	//Условие перехода (20)→(21)
	//Последовательность "Переход К-М" завершена
	IF (K_M.finish) AND drm.timeout THEN
		drm.cmd := drm.error := 0; drm.timer_pt := cycle; drm.inc := FALSE; drm.step := 21;
		btn.K_M.cmd := FALSE; //Шаг проверки: Переход К-М // Кнопка "Переход К-М"
	END_IF;
21:	//Запись уставки таймера шага
	drm.step := 21;//Текущий шаг
	drm.timer_pt := cycle; //Таймер: один цикл вызова

	//Команды текущего шага
	(*1*) btn.NObs.cmd := drm.cmd.0 := drm.step_time <= cycle; //Шаг проверки: АОбс из Магистрали // Кнопка "НОбс"

	//Условие перехода (21)→(22)
	//Последовательность "НОбс" завершена
	IF (NObs.finish) AND drm.timeout THEN
		drm.cmd := drm.error := 0; drm.timer_pt := cycle; drm.inc := FALSE; drm.step := 22;
		btn.NObs.cmd := FALSE; //Шаг проверки: АОбс из Магистрали // Кнопка "НОбс"
	END_IF;
22:	//Запись уставки таймера шага
	drm.step := 22;//Текущий шаг
	drm.timer_pt := cycle; //Таймер: один цикл вызова

	//Команды текущего шага
	(*1*) btn.Bleeding.cmd := drm.cmd.0 := TRUE; //Шаг проверки: Стравливание из ГР под газом // Кнопка "Стравливание ЦБК"

	//Условие перехода (22)→(23)
	//Последовательность "Стравливание" завершена
	IF (Bleeding_full.finish) AND drm.timeout THEN
		drm.cmd := drm.error := 0; drm.timer_pt := cycle; drm.inc := FALSE; drm.step := 23;
		btn.Bleeding.cmd := FALSE; //Шаг проверки: Стравливание из ГР под газом // Кнопка "Стравливание ЦБК"
	END_IF;
23:	//Запись уставки таймера шага
	drm.step := 23;//Текущий шаг
	drm.timer_pt := 10; //Таймер: 10 секунд

	//Команды текущего шага
	(*1*) btn.Repair.cmd := drm.cmd.0 := drm.step_time <= cycle; //Шаг проверки: Переход в Ремонт // Кнопка "Ремонт"

	//Условие перехода (23)→(24)
	//Режим Ремонт
	IF (mde.Repair) AND drm.timeout THEN
		drm.cmd := drm.error := 0; drm.timer_pt := cycle; drm.inc := FALSE; drm.step := 24;
		btn.Repair.cmd := FALSE; //Шаг проверки: Переход в Ремонт // Кнопка "Ремонт"
	END_IF;
24:	//Запись уставки таймера шага
	drm.step := 24;//Текущий шаг
	drm.timer_pt := cycle; //Таймер: один цикл вызова

	//Команды текущего шага
	(*1*) finish := drm.cmd.0 := TRUE; //Завершение
	(*1*) drm.error.0 := NOT btn.test_off.out; //Нажмите кнопку "Комплексное тестирование отключить"

	//Условие перехода (24)→(0)
	//Кнопка "Комплексное тестирование отключить"
	IF (btn.test_off.out) AND drm.timeout THEN
		drm.cmd := drm.error := 0; drm.timer_pt := cycle; drm.inc := FALSE; drm.step := -1;
		finish := FALSE; //Завершение
	END_IF;
END_CASE

//Принудительный выход из последовательности
IF break THEN
	drm.step := -1; drm.cmd := drm.error := 0; drm.timer_pt := cycle; drm.inc := FALSE;
	init := FALSE; //Переинициализирование переменных
	btn.GR.cmd := FALSE; //Шаг проверки: ХП из ГР // Кнопка "ГР"
	btn.HP.cmd := FALSE; //Шаг проверки: ХП из ГР // Кнопка "ХП"
	btn.Start.cmd := FALSE; //Шаг проверки: ХП из ГР // Кнопка "Пуск"
	btn.KPK.cmd := FALSE; //Шаг проверки: КПК из ГР // Кнопка "КПК"
	btn.Start.cmd := FALSE; //Шаг проверки: КПК из ГР // Кнопка "Пуск"
	btn.APK.cmd := FALSE; //Шаг проверки: АПК из ГР под газом // Кнопка "АПК"
	btn.Start.cmd := FALSE; //Шаг проверки: АПК из ГР под газом // Кнопка "Пуск"
	btn.AOss.cmd := FALSE; //Шаг проверки: АОсс из Кольца // Кнопка "АОсс"
	btn.Unlock.cmd := FALSE; //Шаг проверки: АОсс из Кольца // Кнопка "Деблокировка"
	btn.GR.cmd := FALSE; //Шаг проверки: АПК из ГР без газа // Кнопка "ГР"
	btn.APK.cmd := FALSE; //Шаг проверки: АПК из ГР без газа // Кнопка "АПК"
	btn.Start.cmd := FALSE; //Шаг проверки: АПК из ГР без газа // Кнопка "Пуск"
	btn.NOss.cmd := FALSE; //Шаг проверки: НОсс из Кольца // Кнопка "НОсс"
	btn.GR.cmd := FALSE; //Шаг проверки: АПМ из ГР без газа // Кнопка "ГР"
	btn.AObs.cmd := FALSE; //Шаг проверки: АОбс из Магистрали // Кнопка "АОбс"
	btn.Unlock.cmd := FALSE; //Шаг проверки: АОбс из Магистрали // Кнопка "Деблокировка"
	btn.M_K.cmd := FALSE; //Шаг проверки: Переход М-К // Кнопка "Переход М-К"
	cmd_Nst_5000 := FALSE; //Шаг проверки: Повышение Nст до 5000 об/мин
	btn.K_M.cmd := FALSE; //Шаг проверки: Переход К-М // Кнопка "Переход К-М"
	btn.NObs.cmd := FALSE; //Шаг проверки: АОбс из Магистрали // Кнопка "НОбс"
	btn.Bleeding.cmd := FALSE; //Шаг проверки: Стравливание из ГР под газом // Кнопка "Стравливание ЦБК"
	btn.Repair.cmd := FALSE; //Шаг проверки: Переход в Ремонт // Кнопка "Ремонт"
	finish := FALSE; //Завершение
END_IF;

                  
END_FUNCTION_BLOCK

{region INFO}
(*
Назначение: Обновление настроек
Автор     : Дергаев
Дата      : 12.05.2025 16:11:36
Версия    : 00.01.00
*)
{endregion}
FUNCTION FuelRegTuns_update : BOOL
VAR_INPUT
END_VAR
VAR
END_VAR

                    FuelReg.limValUpNvd ();
FuelReg.limValUpNst ();
FuelReg.limValUpTst ();
FuelReg.limValUpTstStart();
FuelReg.limValUpPk ();
FuelReg.RegLimValUpNvd ();
FuelReg.RegLimValDnNvd ();
FuelReg.RegLimValUpNst ();
FuelReg.RegLimValUpTst ();
FuelReg.RegLimValUpTstStart();
FuelReg.RegLimValUpPk ();
FuelReg.ignitionStep ();
FuelReg.ignitionDelay ();
FuelReg.ignitionMaxTime ();
FuelReg.ignitionMaxVal ();
FuelReg.rateOnProg ();
FuelReg.stepOnProg ();
FuelReg.tau1vd ();
FuelReg.tau2vd ();
FuelReg.tau1st ();
FuelReg.tau2st();
FuelReg.tau1Tst ();
FuelReg.tau2Tst ();
FuelReg.tau1Pk ();
FuelReg.tau2Pk ();
FuelReg.dzVd ();
FuelReg.dzSt ();
FuelReg.dzTst ();
FuelReg.dzPk ();
FuelReg.kRVd ();
FuelReg.kLupVd ();
FuelReg.kLdnVd ();
FuelReg.kRst ();
FuelReg.kLupST ();
FuelReg.kLupTst ();
FuelReg.kLupPk ();
FuelReg. kCorrNvd();
FuelReg. kCorrNst();
FuelReg. kCorrTst();
FuelReg. kCorrPk ();
FuelReg.setNvdRegOn ();
FuelReg.setNvdStarterOff ();
FuelReg.setNvdHeat ();
FuelReg.setHeatTime ();
FuelReg.setNvdCool ();
FuelReg.setCoolTime ();
FuelReg.setDTign ();
FuelReg.dNvdUpLim();
FuelReg.dNvdDnLim();
FuelReg.dNstUpLim();
FuelReg.dTstUpLim();
FuelReg.dPkUpLim();
FuelReg.lowTonWork();
FuelReg.delayLowTonWork();
FuelReg.rateOnReg ();

                  
END_FUNCTION

// _^ - ^ _
// Автоматическая проверка защит
// Chekmarev

FUNCTION_BLOCK TAutoCheckShield
VAR_IN_OUT
	start	: BOOL;
END_VAR
VAR
	step	: INT := -1;
	// Проверяемые защиты ( FALSE - не проверена / не успех, TRUE - проверена )
	btn_AOss, 
	btn_AObs,
	AO_PRU,
	AO_BA,
	BEAO,
	SurgeD,
	Vs_D_Av,
	KPV2_wOpen,
	KPV4_wOpen,
	KPV15_wOpen,
	Nst_HH,
	Ntk_Av_HH,
	Nst_flt,
	Tg_inSt_HH,
	Fire_OD,
	Tg1_inSTdistort_HH,
	Tg_inSTflt,
	nIgnition,
	Fire_flt,
	Ntk_nBoost,
	DGdistort,
	Pa_out14_HH,
	BZA_ready_2,
	BZA_alr,
	Pm_TK_An,
	Pm_ST_An,
	Tm_outD_HH,
	Chip_outD,
	Ptg_inDG,
	Pm_Starter_Av,
	Pm_Starter_An,
	dP_F_Pv,
	Ptg_inTRK_LL,
	dPmg_LL,
	Pm_N_An,
	Zs_Nl,
	Kr6_OF_start,
	Causeless_KR1_OF,
	Causeless_KR2_OF,
	Causeless_KR6_OF,
	Causeless_KR10_11
			: BOOL;
			
	crsCurrent	: POINTER TO Tcrs;
	
	callCMD		: BOOL;
	timer		: TON; // Общий таймер
	wd			: TON; // злая собака
END_VAR

                    
IF start AND step = -1 THEN
	step := 5;
	start := FALSE;
	ELSE 
		start := FALSE;
END_IF

CASE step OF
	5:		// btn_AOss
		Reset();
		btn_AOss	:= FALSE;
		crsCurrent 	:= ADR ( crs.btn_AOss );
	6:
		APK_start( _time := T#15S, nextStep := step + 4, cmd := btn.AOss.cmd, checkCRS := btn_AOss );
		
	10:		// btn_AObs
		Reset();
		btn_AObs	:= FALSE;
		crsCurrent	:= ADR ( crs.btn_AObs );
	11:
		APK_start( _time := T#30S, nextStep := step + 4, cmd := btn.AObs.cmd, checkCRS := btn_AObs );
		
	15:		// AO_PRU
		Reset();
		AO_PRU		:= FALSE;
		crsCurrent	:= ADR ( crs.AO_PRU );
	16:
		APK_start( _time := T#29S, nextStep := step + 4, cmd := callCMD, checkCRS := AO_PRU );
		dipar.AO_PRU_1.sim_value := callCMD;
		dipar.AO_PRU_2.sim_value := callCMD;
		
	20:
		Reset();
		AO_BA		:= FALSE;
		crsCurrent	:= ADR ( crs.AO_BA );
	21:
		APK_start( _time := T#15S, nextStep := step + 4, cmd := dipar.AO_BA.sim_value, checkCRS := AO_BA );
		
	25:
		Reset();
		BEAO		:= FALSE;
		crsCurrent	:= ADR ( crs.BEAO );
	26:
		APK_start( _time := T#1S, nextStep := step + 4, cmd := dipar.BEAO.sim_value, checkCRS := BEAO );
		
	30:
		step := 31;
	31:
		step := step + 4;
		
	35:
		Reset();
		SurgeD		:= FALSE;
		crsCurrent	:= ADR ( crs.SurgeD );
	36:
		APK_start( _time := T#15S, nextStep := step + 4, cmd := dipar.SurgeD.sim_value, checkCRS := SurgeD );
		
	40:
		Reset();
		Vs_D_Av		:= FALSE;
		crsCurrent	:= ADR ( crs.Vs_D_Av );
	41:
		APK_start( _time := T#15S, nextStep := step + 4, cmd := dipar.Vs_D_Av.sim_value, checkCRS := Vs_D_Av );
		
	45:
		Reset();
		KPV2_wOpen:= FALSE;
		crsCurrent	:= ADR ( crs.KPV234_wOpen );
	46:
		APK_heat( _time := T#15S, nextStep := step + 4, cmd := callCMD, checkCRS := KPV2_wOpen );
		IF callCMD THEN
			dipar.KPV2_off.sim_value := FALSE;
		END_IF
		
	50: step := 51;		// KPV3
	51: step := 55;
	
	55: Reset();
		KPV4_wOpen	:= FALSE;
		crsCurrent	:= ADR ( crs.KPV234_wOpen );
	56: 
		APK_heat( _time := T#1M, nextStep := step + 4, cmd := callCMD, checkCRS := KPV4_wOpen );
		IF callCMD THEN
			dipar.KPV4_off.sim_value := FALSE;
		END_IF
		
	60:
		Reset();
		KPV15_wOpen	:= FALSE;
		crsCurrent	:= ADR ( crs.KPV15_wOpen );
	61:
		APK_work( _time := T#25S, nextStep := step + 4, cmd := callCMD, checkCRS := KPV15_wOpen );
		IF callCMD THEN
			dipar.KPV5_off.sim_value := FALSE;
		END_IF
		
	65:
		Reset();
		Nst_HH		:= FALSE;
		crsCurrent	:= ADR ( crs.Nst_HH );
	66:
		APK_start( _time := T#15S, nextStep := step + 4, cmd := callCMD, checkCRS := Nst_HH );
		acpar.Nst.sim_value := 9301 * TO_BYTE ( callCMD );
		acpar.Nst.sim_on	:= callCMD;
		
	70:
		Reset();
		Ntk_Av_HH	:= FALSE;
		crsCurrent	:= ADR ( crs.Ntk_Av_HH );
	71:
		APK_start( _time := T#15S, nextStep := step + 4, cmd := callCMD, checkCRS := Ntk_Av_HH );
		acpar.Ntk.sim_value := 8401 * TO_BYTE ( callCMD );	// aipar переписывается в ТР
		acpar.Ntk.sim_on	:= callCMD;		
		
	75:
		Reset();
		Nst_flt		:= FALSE;
		crsCurrent	:= ADR ( crs.Nst_flt );
	76:
		APK_start(_time := T#20S, nextStep := step + 4, cmd := callCMD, checkCRS := Nst_flt );
		aipar.Nst_1.flt_test	:= callCMD;
		aipar.Nst_2.flt_test	:= callCMD;
		
	80:
		Reset();
		Tg_inSt_HH	:= FALSE;
		crsCurrent	:= ADR ( crs.Tg_inST_HH );
	81:
		APK_start( _time := T#15S, nextStep := step + 4, cmd := callCMD, checkCRS := Tg_inSt_HH );
		acpar.Tg_inST.sim_value	:= 671 * TO_BYTE ( callCMD );
		acpar.Tg_inST.sim_on	:= callCMD;
		
	85:
		Reset();
		Fire_OD		:= FALSE;
		crsCurrent	:= ADR ( crs.Fire_OD );
	86:
		APK_start( _time := T#1S, nextStep := step + 4, cmd := dipar.Fire_OD.sim_value, checkCRS := Fire_OD );
		
	90:
		Reset();
		Tg1_inSTdistort_HH	:= FALSE;
		crsCurrent			:= ADR ( crs.Tg1_inSTdistort_HH );
	91:
		APK_heat(_time := T#30S, nextStep := step + 4, cmd := callCMD, checkCRS := Tg1_inSTdistort_HH );
		aipar.Tg_inST_1.sim_value := acpar.Tg_inST.value + 150 * TO_BYTE ( callCMD );
		
	95:
		Reset();
		Tg_inSTflt	:= FALSE;
		crsCurrent	:= ADR ( crs.Tg_inSTflt );
	96:
		APK_start( _time := T#10S, nextStep := step + 4, cmd := callCMD, checkCRS := Tg_inSTflt );
		aipar.Tg_inST_1.flt_test := callCMD;
		aipar.Tg_inST_3.flt_test := callCMD;
		aipar.Tg_inST_5.flt_test := callCMD;
		aipar.Tg_inST_6.flt_test := callCMD;
		
	100:
		Reset();
		nIgnition	:= FALSE;
		crsCurrent	:= ADR ( crs.nIgnition );		
	101:
		APK_start(_time := T#10S, nextStep := step + 4, cmd := callCMD, checkCRS := nIgnition );
		IF am.AZ.on AND callCMD THEN
			am.SK.on := FALSE;
		END_IF
	
	105:
		Reset();
		Fire_flt	:= FALSE;
		crsCurrent	:= ADR ( crs.Fire_flt );
	106:
		APK_work( _time := T#21S, nextStep := step + 4, cmd := callCMD, checkCRS := Fire_flt );
		crs.Tg1_inSTdistort_HH.alg_check := callCMD;
		crs.Tg2_inSTdistort_HH.alg_check := callCMD;
		crs.Tg3_inSTdistort_HH.alg_check := callCMD;
		crs.Tg4_inSTdistort_HH.alg_check := callCMD;
		crs.Tg5_inSTdistort_HH.alg_check := callCMD;
		crs.Tg6_inSTdistort_HH.alg_check := callCMD;
		acpar.Tg_inST.sim_on := callCMD;
		IF callCMD THEN
			acpar.Tg_inST.sim_value := acpar.Tg_inST.value - 10.0;
		END_IF
		
	110:
		Reset();
		Ntk_nBoost	:= FALSE;
		crsCurrent	:= ADR ( crs.Ntk_nBoost );
	111:
		APK_start( _time := T#30S, nextStep := step + 4, cmd := callCMD, checkCRS := Ntk_nBoost );
		acpar.Ntk.sim_on := callCMD AND aipar.Ntk_1.value > 5500;
		acpar.Nst.sim_on := callCMD AND aipar.Nst_1.value > 9100;
		acpar.Ntk.sim_value := 5500;
		acpar.Nst.sim_value := 9000;

	115:
		Reset();
		DGdistort	:= FALSE;
		crsCurrent	:= ADR ( crs.DGdistort );
	116:
		APK_heat( _time := T#10S, nextStep := step + 4, cmd := callCMD, checkCRS := DGdistort );
		aipar.DG_pos.sim_value := aopar.DG_set.value + 2 * TO_BYTE ( callCMD );
		
	120:
		Reset();
		Pa_out14_HH	:= FALSE;
		crsCurrent	:= ADR ( crs.Pa_out14_HH );
	121:
		APK_heat( _time := T#15S, nextStep := step + 4, cmd := callCMD, checkCRS := Pa_out14_HH );
		aipar.Pa_out14.sim_value := 2.1 * TO_BYTE ( callCMD );
		
	125:
		Reset();
		BZA_ready_2	:= FALSE;
		crsCurrent	:= ADR ( crs.BZA_ready_2 );
	126:
		APK_start( _time := T#1S, nextStep := step + 4, cmd := callCMD, checkCRS := BZA_ready_2 );
		IF callCMD THEN
			dipar.BZA_ready_2.sim_value := NOT callCMD;
		END_IF		
	
	130:
		Reset();
		BZA_alr		:= FALSE;
		crsCurrent	:= ADR ( crs.BZA_alr );
	131:
		APK_start( _time := T#45S, nextStep := step + 4, cmd := dipar.BZA_alr.sim_value, checkCRS := BZA_alr );
		
	135:
		Reset();
		Pm_TK_An	:= FALSE;
		crsCurrent	:= ADR ( crs.Pm_TK_An );
	136:
		APK_start( _time := T#1M, nextStep := step + 4, cmd := dipar.Pm_TK_An.sim_value, checkCRS := Pm_TK_An );
		
	140:
		Reset();
		Pm_ST_An	:= FALSE;
		crsCurrent	:= ADR ( crs.Pm_ST_An );
	141:
		APK_start( _time := T#70S, nextStep := step + 4, cmd := dipar.Pm_ST_An.sim_value, checkCRS := Pm_ST_An );
		
	145:
		Reset();
		Tm_outD_HH	:= FALSE;
		crsCurrent	:= ADR ( crs.Tm_outD_HH );
	146:
		APK_heat( _time := T#10S, nextStep := step + 4, cmd := callCMD, checkCRS := Tm_outD_HH );
		aipar.Tm_outD.sim_value	:= 86 * TO_BYTE ( callCMD );
		
	150:
		Reset();
		Chip_outD	:= FALSE;
		crsCurrent	:= ADR ( crs.Chip_outD );
	151:
		APK_start( _time := T#11S, nextStep := step + 4, cmd := dipar.Chip_outD.sim_value, checkCRS := Chip_outD );
		
	155:
		Reset();
		Ptg_inDG	:= FALSE;
		crsCurrent	:= ADR ( crs.Ptg_inDG_An );
	156:
		APK_start( _time := T#1M, nextStep := step + 4, cmd := dipar.Ptg_inDG_An.sim_value, checkCRS := Ptg_inDG );
		
	160:
		Reset();
		Pm_Starter_Av	:= FALSE;
		crsCurrent		:= ADR ( crs.Pm_Starter_Av );
	161:
		APK_start( _time := T#1M, nextStep := step + 4, cmd := callCMD, checkCRS := Pm_Starter_Av );
		dipar.Pm_Starter_Av.sim_value := callCMD;
	
	165:
		Reset();
		Pm_Starter_An	:= FALSE;
		crsCurrent		:= ADR ( crs.Pm_Starter_An );
	166:
		HP( _time := T#70S, nextStep := step + 4, cmd := callCMD, checkCRS := Pm_Starter_An );
		dipar.Pm_Starter_An.sim_value := callCMD;
		
	170:
		Reset();
		dP_F_Pv		:= FALSE;
		crsCurrent	:= ADR ( crs.dP_F_Pv );
	171:
		APK_start( _time := T#15S, nextStep := step + 4, cmd := dipar.dP_F_Pv.sim_value, checkCRS := dP_F_Pv );
	
	175:
		Reset();
		Ptg_inTRK_LL:= FALSE;
		crsCurrent	:= ADR ( crs.Ptg_inTRK_LL );
	176:
		APK_heat( _time := T#15S, nextStep := step + 4, cmd := callCMD, checkCRS := Ptg_inTRK_LL );
		IF callCMD THEN
			aipar.Ptg_inTRK.sim_value := 0.9;
		END_IF
		
	180:
		step := 181;
	181:
		step := step + 4;
		
	185:
		Reset();
		dPmg_LL		:= FALSE;
		crsCurrent	:= ADR ( crs.dPmg_LL );
	186:
		APK_start( _time := T#1M, nextStep := step + 4, cmd := callCMD, checkCRS := dPmg_LL );
		IF callCMD AND aipar.dPmg.value > 0.71 THEN
			aipar.dPmg.sim_value := 0.2;
		END_IF
		
	190:
		Reset();
		Pm_N_An		:= FALSE;
		crsCurrent	:= ADR ( crs.Pm_N_An );
	191:
		APK_start( _time := T#1M, nextStep := step + 4, cmd := dipar.Pm_N_An.sim_value, checkCRS := Pm_N_An );
	
	195:
		Reset();
		Zs_Nl		:= FALSE;
		crsCurrent	:= ADR ( crs.Zs_Nl );
	196:
		APK_start( _time := T#1M, nextStep := step + 4, cmd := dipar.Zs_Nl.sim_value, checkCRS := Zs_Nl );
		
	200:
		step := 201;
	201:
		step := step + 4;
	
	205:
		Reset();
		Kr6_OF_start	:= FALSE;
		crsCurrent		:= ADR ( crs.Kr6_off_start );
	206:
		APK_heat( _time := T#2M, nextStep := step + 4, cmd := callCMD, checkCRS := Kr6_OF_start );
		IF acpar.Nst.value > 300 THEN
			dipar.Kr6_off.sim_value := TRUE;
		END_IF
		
	210:
		Reset();
		Causeless_KR1_OF:= FALSE;
		crsCurrent		:= ADR ( crs.Causeless_KR1_off );
	211:
		APK_work( _time := T#1M, nextStep := step + 4, cmd := callCMD, checkCRS := Causeless_KR1_OF );
		IF callCMD THEN
			dipar.Kr1_ON.sim_value := NOT callCMD;
		END_IF
		
	215:
		Reset();
		Causeless_KR2_OF:= FALSE;
		crsCurrent		:= ADR ( crs.Causeless_KR2_off );
	216:
		APK_work( _time := T#1M, nextStep := step + 4, cmd := callCMD, checkCRS := Causeless_KR2_OF );
		IF callCMD THEN
			dipar.Kr2_ON.sim_value := NOT callCMD;
			dipar.Kr6_off.sim_value := callCMD;
		END_IF
		
	220:
		Reset();
		Causeless_KR6_OF := FALSE;
		crsCurrent		:= ADR ( crs.Causeless_KR6_off );
	221: 
		APK_work( _time := T#1M, nextStep := step + 4, cmd := callCMD, checkCRS := Causeless_KR6_OF );
		IF callCMD THEN
			dipar.Kr2_off.sim_value := callCMD;
			dipar.Kr6_ON.sim_value := NOT callCMD;
		END_IF
		
	225:
		Reset();
		Causeless_KR10_11:= FALSE;
		crsCurrent		:= ADR( crs.Causeless_KR10_11 );
	226:
		APK_start( _time := T#5M, nextStep := step + 4, cmd := callCMD, checkCRS := Causeless_KR10_11 );
		IF am.Kr15.on THEN
			dipar.Kr10_off.sim_value := FALSE;
		END_IF
		
	230:
		step := -1;
	
END_CASE

timer();
                  

ACTION Reset:
                        
timer ( IN := ( AOss.break XOR AOss.finish ) AND ( AObs.break XOR AObs.finish ) AND NOT timer.Q, PT := T#5S );
btn.Unlock.cmd 	:= timer.Q;
btn.GR.cmd		:= AOss.break AND aobs.break;
IF mde.GR THEN
	timer ( IN := FALSE );
	step := step + 1;
END_IF
wd ( IN := FALSE );
                      
END_ACTION

METHOD PRIVATE APK_start : BOOL
VAR_INPUT
	_time	: TIME;
	nextStep: INT;
END_VAR
VAR_IN_OUT
	cmd		: BOOL;
	checkCRS: BOOL;
END_VAR
                          IF mde.GR THEN
	timer (IN := TRUE, PT := T#5S);
	btn.APK.cmd := timer.Q;
END_IF
IF tch.ReadyAPK.value THEN
	timer ( IN := FALSE );
	btn.Unlock.cmd 	:= TRUE;
	btn.Start.cmd	:= TRUE;
END_IF
IF mde.APK THEN
	timer (IN := TRUE, PT := _time);
	cmd := timer.Q;
END_IF		
IF crsCurrent^.out THEN
	timer (IN 	:= FALSE);
	checkCRS 	:= TRUE;
	cmd			:= FALSE;
	step := nextStep;
	wd ( IN := FALSE );
END_IF

wd ( IN := TRUE, PT := T#5M + _time );
IF wd.Q THEN
	btn.AObs.cmd := TRUE;
	step 	:= nextStep;
	cmd		:= FALSE;
END_IF
                        
END_METHOD

METHOD PRIVATE APK_heat : BOOL
VAR_INPUT
	_time	: TIME;
	nextStep: INT;
END_VAR
VAR_IN_OUT
	cmd		: BOOL;
	checkCRS: BOOL;
END_VAR
                          IF mde.GR THEN
	timer (IN := TRUE, PT := T#5S);
	btn.APK.cmd := timer.Q;
END_IF
IF tch.ReadyAPK.value THEN
	timer (IN := FALSE);
	btn.Unlock.cmd 	:= TRUE;
	btn.Start.cmd	:= TRUE;
END_IF
IF tch.GTDHeat.value THEN
	timer (IN := TRUE, PT := _time);
	cmd := timer.Q;
END_IF		
IF crsCurrent^.out THEN
	timer (IN 	:= FALSE);
	checkCRS 	:= TRUE;
	cmd			:= FALSE;
	step := nextStep;
	wd ( IN := FALSE );
END_IF

wd ( IN := TRUE, PT := T#10M );
IF wd.Q THEN
	btn.AObs.cmd := TRUE;
	step 	:= nextStep;
	cmd		:= FALSE;
END_IF
                        
END_METHOD

METHOD PRIVATE APK_work : BOOL
VAR_INPUT
	_time	: TIME;
	nextStep: INT;
END_VAR
VAR_IN_OUT
	cmd		: BOOL;
	checkCRS: BOOL;
END_VAR
                          IF mde.GR THEN
	timer (IN := TRUE, PT := T#5S);
	btn.APK.cmd := timer.Q;
END_IF
IF tch.ReadyAPK.value THEN
	timer (IN := FALSE);
	btn.Unlock.cmd 	:= TRUE;
	btn.Start.cmd	:= TRUE;
END_IF
IF tch.GTDwork.value THEN
	timer (IN := TRUE, PT := _time);
	cmd := timer.Q;
END_IF		
IF crsCurrent^.out THEN
	timer (IN 	:= FALSE);
	checkCRS 	:= TRUE;
	cmd			:= FALSE;
	step := nextStep;
	wd ( IN := FALSE );
END_IF

wd ( IN := TRUE, PT := T#10M + _time );
IF wd.Q THEN
	btn.AObs.cmd := TRUE;
	step 	:= nextStep;
	cmd		:= FALSE;
END_IF
                        
END_METHOD

METHOD PRIVATE HP : BOOL
VAR_INPUT
	_time	: TIME;
	nextStep: INT;
END_VAR
VAR_IN_OUT
	cmd		: BOOL;
	checkCRS: BOOL;
END_VAR
                          IF mde.GR THEN
	timer (IN := TRUE, PT := T#5S);
	btn.HP.cmd := timer.Q;
END_IF
IF tch.ReadyHP.value THEN
	timer (IN := FALSE);
	btn.Unlock.cmd 	:= TRUE;
	btn.Start.cmd	:= TRUE;
END_IF
IF mde.HP THEN
	timer (IN := TRUE, PT := _time);
	cmd := timer.Q;
END_IF
IF crsCurrent^.out THEN
	timer (IN 	:= FALSE);
	checkCRS 	:= TRUE;
	cmd			:= FALSE;
	step := nextStep;
	wd ( IN := FALSE );
END_IF
wd ( IN := TRUE, PT := T#3M );
IF wd.Q THEN
	btn.AObs.cmd := TRUE;
	step 	:= nextStep;
	cmd		:= FALSE;
END_IF
                        
END_METHOD
END_FUNCTION_BLOCK

FUNCTION fun_ACS : BOOL
VAR_INPUT
END_VAR
VAR
END_VAR

                    ACS.ACS ( start := ACS.startACS );
                  
END_FUNCTION

{region INFO}
(*
 Назначение: Используется для присвоения переменным, предназначенным для передачи по МЭК-104 соответствующих значений
 Автор:      /Andrey/ 16.07.2025 17:15:07
*)
{endregion}
FUNCTION IEC104_update : BOOL
VAR_INPUT
END_VAR
VAR
END_VAR

                    //Режим/Тип:int4/Адрес:1
IEC104.GVL_mde_hmi_number.value := GVL.mde_hmi.number;
//Тест: пила, базовый цикл/Тип:REAL/Адрес:2
IEC104.test_Saw_Slow_value.value := test.Saw_Slow.value;
//Тест: пила, быстрый цикл/Тип:REAL/Адрес:3
IEC104.test_Saw_Fast_value.value := test.Saw_Fast.value;
//Тест: синус, базовый цикл/Тип:REAL/Адрес:4
IEC104.test_Sin_Slow_value.value := test.Sin_Slow.value;
//Частота вращения ротора ТК (1)/Тип:REAL/Адрес:5
IEC104.aipar_NTK_1_in_value.value := aipar.NTK_1.in_value;
//Частота вращения ротора ТК (2)/Тип:REAL/Адрес:6
IEC104.aipar_NTK_2_in_value.value := aipar.NTK_2.in_value;
//Частота вращения ротора СТ (1)/Тип:REAL/Адрес:7
IEC104.aipar_NST_1_in_value.value := aipar.NST_1.in_value;
//Частота вращения ротора СТ (2)/Тип:REAL/Адрес:8
IEC104.aipar_NST_2_in_value.value := aipar.NST_2.in_value;
//Положение дозирующей иглы ДУС/Тип:REAL/Адрес:9
IEC104.aipar_DG_Pos_in_value.value := aipar.DG_Pos.in_value;
//Давление воздуха за 14-й ступенью осевого компрессора/Тип:REAL/Адрес:10
IEC104.aipar_Pa_out14_in_value.value := aipar.Pa_out14.in_value;
//dP на конфузоре/Тип:REAL/Адрес:11
IEC104.aipar_dP_conf_in_value.value := aipar.dP_conf.in_value;
//Управление ТРК/Тип:REAL/Адрес:12
IEC104.aopar_DG_Set_value.value := aopar.DG_Set.value;
//СК закрыт/Тип:uint4/Адрес:13
IEC104.dipar_SK_off_status.value := dipar.SK_off.status;
//Открыть СК/Тип:uint4/Адрес:14
IEC104.dopar_SK_ON_status.value := dopar.SK_ON.status;
//диаг. (Сигнал управления положением дозатора газа)/Тип:REAL/Адрес:15
IEC104.aipar_DG_Pos_diag_in_value.value := aipar.DG_Pos_diag.in_value;
//Открыть КПВ1, 5/Тип:uint4/Адрес:16
IEC104.dopar_KPV15_ON_status.value := dopar.KPV15_ON.status;

                  
END_FUNCTION

{region INFO}
(*
 Назначение:   Ручной вызов обработчиков дискретных ИМов в base цикле
 Автор:        /chekmarev/ 17.04.2025
 Проект:       KA107
*)
{endregion}
FUNCTION am_update_base : BOOL
VAR
	KPV15du	: BOOL;
	KPV15on	: BOOL;
	KPV15off: BOOL;
	KPV23du	: BOOL;
	KPV23on	: BOOL;
	KPV23off: BOOL;
END_VAR

                    // ---------- блок самоподхвата ДУ у КПВ2 и КПВ3 по изменению одного из них с HMI
KPV23du	:= am.KPV2.cmd.0 OR am.KPV3.cmd.0;	// делаем так, чтобы не плодить глобальные переменные
KPV23on := am.KPV2.cmd.1 OR am.KPV3.cmd.1;
KPV23off := am.KPV2.cmd.2 OR am.KPV3.cmd.2;

engine.KPV2du( in	:= am.KPV2.cmd.0 );		// к этому моменту OPC сервер должен внести изменения в бит, если есть воздействие с HMI
engine.KPV2on( in	:= am.KPV2.cmd.1 );
engine.KPV2off( in	:= am.KPV2.cmd.2 );
engine.KPV3du( in	:= am.KPV3.cmd.0 );
engine.KPV3on( in	:= am.KPV3.cmd.1 );
engine.KPV3off( in	:= am.KPV3.cmd.2 );

IF engine.KPV2du.Qf OR engine.KPV3du.Qf THEN
	KPV23du := TRUE;
END_IF
IF engine.KPV2on.Qf OR engine.KPV3on.Qf THEN
	KPV23on := TRUE;
END_IF
IF engine.KPV2off.Qf OR engine.KPV3off.Qf THEN
	KPV23off := TRUE;
END_IF
IF engine.KPV2du.Qr OR engine.KPV3du.Qr THEN
	KPV23du	:= FALSE;
END_IF
IF engine.KPV2on.Qr OR engine.KPV3on.Qr THEN
	KPV23on := FALSE;
END_IF
IF engine.KPV2off.Qr OR engine.KPV3off.Qr THEN
	KPV23off := FALSE;
END_IF

// ---------- блок самоподхвата ДУ у КПВ1 и КПВ5 по изменению одного из них с HMI
KPV15du	:= am.KPV1.cmd.0 OR am.KPV5.cmd.0;
KPV15on	:= am.KPV1.cmd.1 OR am.KPV5.cmd.1;
KPV15off:= am.KPV1.cmd.2 OR am.KPV5.cmd.2;

engine.KPV1du( in	:= am.KPV1.cmd.0 );
engine.KPV1on( in	:= am.KPV1.cmd.1 );
engine.KPV1off( in	:= am.KPV1.cmd.2 );
engine.KPV5du( in	:= am.KPV5.cmd.0 );
engine.KPV5on( in	:= am.KPV5.cmd.1 );
engine.KPV5off( in	:= am.KPV5.cmd.2 );

IF engine.KPV1du.Qf OR engine.KPV5du.Qf THEN
	KPV15du := TRUE;
END_IF
IF engine.KPV1on.Qf OR engine.KPV5on.Qf THEN
	KPV15on := TRUE;
END_IF
IF engine.KPV1off.Qf OR engine.KPV5off.Qf THEN
	KPV15off := TRUE;
END_IF
IF engine.KPV1du.Qr OR engine.KPV5du.Qr THEN
	KPV15du	:= FALSE;
END_IF
IF engine.KPV1on.Qr OR engine.KPV5on.Qr THEN
	KPV15on := TRUE;
END_IF
IF engine.KPV1off.Qr OR engine.KPV5off.Qr THEN
	KPV15off := TRUE;
END_IF
// -----------------------------------

//КПВ 1
//Тип: 1x2
am.KPV1.cmd.0 	:= KPV15du;
am.KPV1.cmd.1 	:= KPV15on;
am.KPV1.cmd.2 	:= KPV15off;
am.KPV1(
	DU_prm := alg.V_000,
	onSigFlt := dipar.KPV1_ON.flt,
	onSig := dipar.KPV1_ON.value,
	onSig_sim_on := dipar.KPV1_ON.sim_on,
	onSig_sim_value := dipar.KPV1_ON.sim_value,
	offSigFlt := dipar.KPV1_off.flt,
	offSig := dipar.KPV1_off.value,
	offSig_sim_on := dipar.KPV1_off.sim_on,
	offSig_sim_value := dipar.KPV1_off.sim_value,
	onFlt := dopar.KPV15_ON.flt);
// dopar.KPV15_ON.value	-> Вызов в am_update_fast()	
//--------------------------------------------------------------------------

//КПВ 2
//Тип: 1x2
am.KPV2.cmd.0	:= KPV23du;
am.KPV2.cmd.1	:= KPV23on;
am.KPV2.cmd.2	:= KPV23off;
am.KPV2(
	DU_prm := alg.V_000,
	onSigFlt := dipar.KPV2_ON.flt,
	onSig := dipar.KPV2_ON.value,
	onSig_sim_on := dipar.KPV2_ON.sim_on,
	onSig_sim_value := dipar.KPV2_ON.sim_value,
	offSigFlt := dipar.KPV2_off.flt,
	offSig := dipar.KPV2_off.value,
	offSig_sim_on := dipar.KPV2_off.sim_on,
	offSig_sim_value := dipar.KPV2_off.sim_value,
	onFlt := dopar.KPV23_OFF.flt);
//--------------------------------------------------------------------------

//КПВ 3
//Тип: 1x2
am.KPV3.cmd.0	:= KPV23du;
am.KPV3.cmd.1	:= KPV23on;
am.KPV3.cmd.2	:= KPV23off;
am.KPV3(
	DU_prm := alg.V_000,
	onSigFlt := dipar.KPV3_ON.flt,
	onSig := dipar.KPV3_ON.value,
	onSig_sim_on := dipar.KPV3_ON.sim_on,
	onSig_sim_value := dipar.KPV3_ON.sim_value,
	offSigFlt := dipar.KPV3_off.flt,
	offSig := dipar.KPV3_off.value,
	offSig_sim_on := dipar.KPV3_off.sim_on,
	offSig_sim_value := dipar.KPV3_off.sim_value,
	onFlt := dopar.KPV23_OFF.flt);
dopar.KPV23_OFF.value := NOT am.KPV2.onOUT OR NOT am.KPV3.onOut;
//--------------------------------------------------------------------------

// КПВ4
// Штатный вызов (создан конфигуратором)

//КПВ 5
//Тип: 1x2
am.KPV5.cmd.0 := KPV15du;
am.KPV5.cmd.1 := KPV15on;
am.KPV5.cmd.2 := KPV15off;
am.KPV5(
	DU_prm := alg.V_000,
	onSigFlt := dipar.KPV5_ON.flt,
	onSig := dipar.KPV5_ON.value,
	onSig_sim_on := dipar.KPV5_ON.sim_on,
	onSig_sim_value := dipar.KPV5_ON.sim_value,
	offSigFlt := dipar.KPV5_off.flt,
	offSig := dipar.KPV5_off.value,
	offSig_sim_on := dipar.KPV5_off.sim_on,
	offSig_sim_value := dipar.KPV5_off.sim_value,
	onFlt := dopar.KPV15_ON.flt);
// dopar.KPV15_ON.value	-> Вызов в am_update_fast()
//--------------------------------------------------------------------------

//Кран 9
//Тип: 2x2
am.Kr9(
	DU_prm := FALSE,
	onSigFlt := dipar.Kr9_ON.flt,
	onSig := dipar.Kr9_ON.value,
	onSig_sim_on := dipar.Kr9_ON.sim_on,
	onSig_sim_value := dipar.Kr9_ON.sim_value,
	offSigFlt := dipar.Kr9_off.flt,
	offSig := dipar.Kr9_off.value,
	offSig_sim_on := dipar.Kr9_off.sim_on,
	offSig_sim_value := dipar.Kr9_off.sim_value,
	onFlt := dopar.Kr12_ON.flt,
	offFlt := dopar.KR12_OFF.flt);
	
//Кран 10
//Тип: 2x2
am.Kr10(
	DU_prm := FALSE,
	onSigFlt := dipar.Kr10_ON.flt,
	onSig := dipar.Kr10_ON.value,
	onSig_sim_on := dipar.Kr10_ON.sim_on,
	onSig_sim_value := dipar.Kr10_ON.sim_value,
	offSigFlt := dipar.Kr10_off.flt,
	offSig := dipar.Kr10_off.value,
	offSig_sim_on := dipar.Kr10_off.sim_on,
	offSig_sim_value := dipar.Kr10_off.sim_value,
	onFlt := dopar.Kr11_ON.flt,
	offFlt := dopar.Kr11_OFF.flt);
	
// ---------- блок самоподхвата ДУ у КПВ2 и КПВ3 по изменению одного из них с HMI
// выходы триггера сброшены, запоминаем текущее значение
engine.KPV2du( in	:= am.KPV2.cmd.0 );
engine.KPV2on( in	:= am.KPV2.cmd.1 );
engine.KPV2off( in	:= am.KPV2.cmd.2 );
engine.KPV3du( in	:= am.KPV3.cmd.0 );
engine.KPV3on( in	:= am.KPV3.cmd.1 );
engine.KPV3off( in	:= am.KPV3.cmd.2 );
// ------------------------------------
// ---------- блок самоподхвата ДУ у КПВ1 и КПВ5 по изменению одного из них с HMI
engine.KPV1du( in	:= am.KPV1.cmd.0 );
engine.KPV1on( in	:= am.KPV1.cmd.1 );
engine.KPV1off( in	:= am.KPV1.cmd.2 );
engine.KPV5du( in	:= am.KPV5.cmd.0 );
engine.KPV5on( in	:= am.KPV5.cmd.1 );
engine.KPV5off( in	:= am.KPV5.cmd.2 );
// -----------------------------------
                  
END_FUNCTION

FUNCTION AS_Link : BOOL
VAR_INPUT
END_VAR
VAR
END_VAR

                    s_tunpar.ASprot.Pin.value	:= aipar.Pg_inN.value; 
s_tunpar.ASprot.Pout.value	:= aipar.Pg_outN.value; 
s_tunpar.ASprot.Tin.value	:= aipar.Tg_inN.value;  
s_tunpar.ASprot.Tout.value	:= aipar.Tg_outN.value; 
s_tunpar.ASprot.dPconf.value:= aipar.dP_conf.value; 
s_tunpar.ASprot.Nst.value	:= acpar.Nst.value; 
s_tunpar.ASprot.Patm.value	:= 101.6; 

s_tunpar.ASprot.Pin.flt		:= aipar.Pg_inN.flt; 
s_tunpar.ASprot.Pout.flt	:= aipar.Pg_outN.flt; 
s_tunpar.ASprot.Tin.flt		:= aipar.Tg_inN.flt;  
s_tunpar.ASprot.Tout.flt	:= aipar.Tg_outN.flt; 
s_tunpar.ASprot.dPconf.flt	:= TRUE; //aipar.dP_conf.flt; 
s_tunpar.ASprot.Nst.flt		:= acpar.Nst.flt; 

s_tunpar_update();

s_tunpar.ASprot(
	cycle			:= cycle_time_fast, 
	D				:= 0.5917, // относительная плотность газа по воздуху - обычно выход блока расчета газовых констант, для упрощенного проекта задана постоянная
	mu				:= 17.091, // молярная масса газа, кг/кмоль - обычно выход блока расчета газовых констант, для упрощенного проекта задана постоянная
	sigDKS			:= FALSE, // при TRUE сигнал 
	sigPreSurgeOR	:= TRUE, // при TRUE сигнал предпомпажа (защиты) формируется при падении dPk ИЛИ росте Nst, при FALSE при падении dPk И росте Nst, проверить в работе
	protectOn		:= mde.M, // Взведение помпажной защиты. Магистраль? Переход К->М?
	sigCheck		:= mde.PZ, // Проверка защит 
	reset			:= btn.Unlock.out, // Деблокировка 
	calcSRon		:= TRUE,
	sigDKS 			:= TRUE,
	initSecResToMain := 3.0,
 	prod        => s_aspar.prod.value,  // объемная производительность, м3/с
 	prodCom     => s_aspar.prodCom.value, // коммерческая производительность, млн·нм3/сут
  	Qc          => s_aspar.Qc.value, // коммерческая производительность, нм3/ч
  	pressRatio  => s_aspar.pressRatio.value,
  	NstNorm     => s_aspar.NstNorm.value,
 // 	antisurgeBrk=> ,
 // 	mainContBrk => ,
 // 	res1ContBrk => ,
 // 	res2ContBrk => ,
  	surgeRes    => s_aspar.surgeRes.value,
  	ddPconf     => s_aspar.ddPconf.value, // производная перепада давления на конфузоре нагнетателя по времени
  	dNst        => s_aspar.dNst.value, // производная частоты вращения ротора нагнетателя по времени
  	preSurge    => tch.AS_preSurge.value, // сигнал "Предпомпажное состояние"
 	surge       => tch.AS_surge.value, // сигнал "Помпаж нагнетателя"
 // 	surgeAlertBrk=> , // сигнал "Отказ сигнализатора помпажа"
  	surgeSign_ddPconf=> tch.AS_surgeSign_ddPconf.value, // внутренний сигнал "Предпомпажное состояние" по падению dP на конфузоре //Dergaev 2024-11-02
  	surgeSign_dNst	=> tch.AS_surgeSign_dNst.value // внутренний сигнал "Предпомпажное состояние" по росту частоты вращения  //Dergaev 2024-11-02

//	emergOpenBypass=> Команда на 6 (вход в обработчик ИМ) - см. ALG_GO_AM
    
   );
   
 s_tunpar.ASprot.update();  
                  
END_FUNCTION

FUNCTION_BLOCK TASProtector
VAR_INPUT
// время цикла
  cycle : REAL;

// входные аналоговые параметры
  Pin    : Taspar; // P газа на входе ЦБК, МПа
  Pout   : Taspar; // P газа на выходе ЦБК, МПа
  Tin    : Taspar; // T газа на входе ЦБК, °С
  Tout   : Taspar; // T газа на выходе ЦБК, °С
  dPconf : Taspar; // перепад давления на конфузоре, кПа
  Nst    : Taspar; // Частота вращения СТ, об/мин
  Patm   : Taspar; // атмосферное давление, кПа
  
  D				: REAL; // относительная плотность газа по воздуху
  mu			: REAL; // молярная масса газа, кг/кмоль

  sigDKS        : BOOL; // работа на ДКС/линейной  КС
  sigPreSurgeOR : BOOL; // условие формировани¤ предпомпажного состо¤ни¤  
  protectOn 	: BOOL; // включить защиту
  sigCheck      : BOOL; // проверка защит
  reset			: BOOL; // сброс триггера открытия	
  check 		: BOOL; // проверка защит 
  calcSRon		: BOOL; // расчет помпажного запаса использовать
  initSecResToMain : REAL := 1.0; // начальное значение коэффициента пересчета второго контура в основной
END_VAR
VAR_OUTPUT
  prod        : REAL := 0.0 ; // объемная производительность, м3/с
  prodCom     : REAL := 0.0 ; // коммерческая производительность, млн·нм3/сут
  Qc          : REAL := 0.0 ; // коммерческая производительность, нм3/ч
  pressRatio  : REAL := 1.0 ;
  NstNorm     : REAL := 0.0 ;
  antisurgeBrk: BOOL := FALSE;
  mainContBrk : BOOL := false;
  res1ContBrk : BOOL := false;
  res2ContBrk : BOOL := false;
  surgeRes    : REAL := 100.0;
  ddPconf       : REAL; // производная перепада давления на конфузоре нагнетателя по времени
  dNst          : REAL; // производная частоты вращения ротора нагнетателя по времени
  preSurge      : BOOL; // сигнал "Предпомпажное состояние"
  surge         : BOOL; // сигнал "Помпаж нагнетателя"
  surgeAlertBrk : BOOL; // сигнал "Отказ сигнализатора помпажа"
  surgeSign_ddPconf : BOOL; // внутренний сигнал "Предпомпажное состояние" по падению dP на конфузоре //Dergaev 2024-11-02
  surgeSign_dNst	: BOOL; // внутренний сигнал "Предпомпажное состояние" по росту частоты вращения  //Dergaev 2024-11-02

  emergOpenBypass : BOOL; // команда экстренного открытия байпаса	
END_VAR
VAR
  resCalc      	: TSurgeResCalc; // блок расчета помпажного запаса
  surgeAlert   	: TSurgeAlert  ; // блок диагностики предпомпажного состояния
  init			: BOOL := TRUE; 	
END_VAR

                    
                  

METHOD update : BOOL
VAR_INPUT
END_VAR
                          // вычислить помпажный запас
resCalc(cycle  := cycle,
            Nst    := Nst.value,
            Pin    := Pin.value,
            Pout   := Pout.value,
            Tin    := Tin.value,
            dPconf := dPconf.value,
            Patm   := Patm.value,
            NstBrk    := Nst.flt,
            PinBrk    := Pin.flt,
            PoutBrk   := Pout.flt,
            dPconfBrk := dPconf.flt,
            c2Main := s_tunpar.c2Main.value,
            c1Main := s_tunpar.c1Main.value,
            c0Main := s_tunpar.c0Main.value,
            c21Res := s_tunpar.c2Res1.value,
            c11Res := s_tunpar.c1Res1.value,
            c01Res := s_tunpar.c0Res1.value,
            c22Res := s_tunpar.c2Res2.value,
            c12Res := s_tunpar.c1Res2.value,
            c02Res := s_tunpar.c0Res2.value,
            kConf  := s_tunpar.Kconf.value,
            nNorm  := s_tunpar.nNorm.value,
            D      := D,
            mu     := mu,
            check  := sigCheck,
			initSecResToMain := initSecResToMain,
			NstNorm=>NstNorm , 
			antisurgeBrk=>antisurgeBrk , 
			mainContBrk=>mainContBrk , 
			res1ContBrk=>res1ContBrk , 
			res2ContBrk=>res2ContBrk  );

IF protectOn THEN
	prod:=resCalc.prod; 
	prodCom:=resCalc.prodCom; 
	Qc:=resCalc.Qc; 
	pressRatio:=resCalc.pressRatio;
	surgeRes:=resCalc.surgeRes; 
ELSE
	prod:=0.0; 
	prodCom:=0.0; 
	Qc:=0.0; 
	pressRatio:=1.0; 			
	surgeRes:=100.0; 
END_IF;			
// обновить сигнализатор помпажа
surgeAlert( dPconf        := dPconf.value,
          	Nst           := Nst.value,
            dPconfBrk     := dPconf.flt,
          	NstBrk        := Nst.flt,
          	maxRateDPconf := s_tunpar.maxRateDPconf.value,
          	maxRateNst    := s_tunpar.maxRateNst.value,
          	SAoffDelay    := s_tunpar.SAoffDelay.value,
          	SAdelay       := s_tunpar.SAdelay.value,
          	blockDelay    := s_tunpar.blockDelay.value,
          	resetDelay    := s_tunpar.resetDelay.value,
          	cycle         := cycle,
          	permit        := protectOn,
          	alternate     := sigDKS,
          	preSurgeOR    := sigPreSurgeOR,
          	init          := init,
          	check         := sigCheck,
			ddPconf=>ddPconf , 
			dNst=>dNst , 
			preSurge=>preSurge , 
			surge=>surge , 
			surgeAlertBrk=>surgeAlertBrk , 
			surgeSign_ddPconf=>surgeSign_ddPconf , 
			surgeSign_dNst=>surgeSign_dNst );
			
IF init THEN init := FALSE; END_IF;			

// принудительное открытие байпаса
emergOpenBypass :=  protectOn AND NOT check AND ( surgeAlert.preSurge OR surgeAlert.surge OR calcSRon AND ( resCalc.surgeRes < s_tunpar.minSR.value ) OR emergOpenBypass ) AND NOT reset;
                        
END_METHOD
END_FUNCTION_BLOCK

{region INFO}
(*
Назначение: Числовые настройки
Автор     : Дергаев
Дата      : 20.03.2025 16:19:20
Версия    : 00.00.02
*)
{endregion}
FUNCTION s_tunpar_update : BOOL
VAR_INPUT
END_VAR
VAR
END_VAR

                    // код для функции обновления настроек
s_tunpar.c2Main(); // Коэфф. при 2-й степ. осн. системы координат
s_tunpar.c1Main(); // Коэфф. при 1-й степ. осн. системы координат
s_tunpar.c0Main(); // Коэфф. при 0-й степ. осн. системы координат
s_tunpar.c2Res1(); // Коэфф. при 2-й степ. 1-й рез. системы координат
s_tunpar.c1Res1(); // Коэфф. при 1-й степ. 1-й рез. системы координат
s_tunpar.c0Res1(); // Коэфф. при 0-й степ. 1-й рез. системы координат
s_tunpar.c2Res2(); // Коэфф. при 2-й степ. 2-й рез. системы координат
s_tunpar.c1Res2(); // Коэфф. при 1-й степ. 2-й рез. системы координат
s_tunpar.c0Res2(); // Коэфф. при 0-й степ. 2-й рез. системы координат
s_tunpar.minSR(); // Мин. помпажный запас
s_tunpar.maxPout (); // Макс. давление на выходе Н
s_tunpar.maxPR (); // Макс. степень сжатия
s_tunpar.Kconf(); // Коэффициент конфузора
s_tunpar.nNorm (); // Номинальная N СТ
s_tunpar.maxRateDPconf (); // Макс. ск. падения dP на конфузоре
s_tunpar.maxRateNst (); // Макс. ск. нарастания N СТ
s_tunpar.maxRateSR(); // Макс. ск. падения помпажного запаса
s_tunpar.maxRateSR_KM(); // Макс. ск. падения помпажного запаса К->М

                  
END_FUNCTION

FUNCTION handleMotoClock : BOOL

                    MotoClockGPA(
				start 	:= am.SK.on,
				stop	:= NOT am.SK.on,
				NO		:= alg.NO,
				AO		:= alg.AO,
				work	:= tch.GTDwork.value,
				reserve	:= alg.V_000,
				gaz		:= tch.Gas_N.value,
				
				countStart 	:= tunpar.countStart,
				countNO		:= tunpar.countNO,
				countAO		:= tunpar.countAO,
				generalOpTime	:= tunpar.generalOpTime,
				workOpTime		:= tunpar.workOpTime );
                  
END_FUNCTION

// Класс, обслуживающий наработку агрегата, а также подсчёт пуско-остановов
// Chekmarev
{attribute 'symbol' := 'none'}
FUNCTION_BLOCK TMotoClockHandler
VAR_INPUT
	start		: BOOL;		// сигнал пуска агрегата
	stop		: BOOL;		// сигнал останова двигателя
	NO			: BOOL;		// сигнал НО
	AO			: BOOL;		// сигнал АО
	work		: BOOL;		// агрегат в работе
	reserve		: BOOL;		// агрегат в резерве/ремонте
	gaz			: BOOL;		// газ в контуре
	path		: STRING := 'OpTime/engine/count.txt';	// путь до файла
END_VAR
VAR
	Qstart			: TEdgeDetect;
	Qno				: TEdgeDetect;
	Qao				: TEdgeDetect;
	
	// экземпляр ФБ для работы с файлом счётчиков пусков/остановов
	countFile	: FileManager;
	// ошибка работы с файлом
	err			: INT;
	init		: BOOL;
	// признак необходимости записи значений в файл
	xWrite		: BOOL;
	// признак пуска двигателя
	isStarted	: BOOL;
	// прежнее время
	oldTime		: UDINT;
	// временные переменные для хранения наработок
	generalOpTimeTemp,
	generalOpTimeOld,
	workOpTimeTemp,
	workOpTimeOld	: REAL;
END_VAR
VAR_IN_OUT
	// количество пусков
	countStart	: Ttunpar;
	// количество НО
	countNO		: Ttunpar;
	// количество АО
	countAO		: Ttunpar;

	// общая наработка в часах
	generalOpTime: Ttunpar;
	// наработка на режиме в часах
	workOpTime	: Ttunpar;
END_VAR
VAR CONSTANT
	rn	: STRING := '$R$N';
END_VAR

                    
Qstart( in := start );
Qno( in := NO );
Qao( in := AO );

IF Qstart.Qf THEN
	countStart.value := countStart.value + 1;
	xWrite := TRUE;
END_IF

IF Qno.Qr AND NOT AO THEN
	countNO.value	:= countNO.value + 1;
	xWrite := TRUE;
END_IF

IF Qao.Qf AND ( NOT reserve OR gaz ) THEN
	countAO.value	:= countAO.value + 1;
	xWrite := TRUE;
END_IF

IF NOT init THEN
	countFile.FileName := path;
	init := Read();
END_IF

IF xWrite THEN
	xWrite := NOT Write();
END_IF

countFile.Update();

isStarted := ( start OR isStarted ) AND NOT stop;
xWrite := OpTime();
                  

METHOD PRIVATE Write : BOOL
VAR
	temp	: STRING;
END_VAR
                          IF NOT countfile.xBusy THEN
	temp := CONCAT( TO_STRING( countStart.value ), rn );
	temp := CONCAT( temp, TO_STRING( countNO.value ));
	temp := CONCAT( temp, rn );
	temp := CONCAT( temp, TO_STRING( countAO.value ));
	temp := CONCAT( temp, rn );
	temp := CONCAT( temp, TO_STRING( generalOpTime.value ));
	temp := CONCAT( temp, rn );
	temp := CONCAT( temp, TO_STRING( workOpTime.value ));

	countFile.Record := temp;
END_IF

IF countFile.WDone THEN
	Write := TRUE;
END_IF

IF countFile.xError THEN
	err := countFile.eError;
	Write := TRUE;
END_IF
                        
END_METHOD

METHOD PRIVATE Read : BOOL
VAR
	temp	: STRING;
	sstart,
	sNO,
	sAO,
	sGeneral,
	sWork	: STRING;
	
	pos		: INT;
	l		: INT;
END_VAR
                          temp := countFile.Record;

IF countFile.RDone THEN
	pos		:= FIND( temp, rn ) - 1;
	sstart 	:= LEFT( temp, pos );
	pos 	:= pos + LEN( rn );
	temp	:= RIGHT( temp, LEN( temp ) - pos );
	pos 	:= FIND( temp , rn )- 1;
	sNO		:= LEFT( temp, pos );
	pos		:= pos + LEN( rn );
	temp	:= RIGHT( temp, LEN( temp ) - pos );
	pos		:= FIND( temp, rn ) - 1;
	sAO		:= LEFT( temp, pos );
	pos		:= pos + LEN( rn );
	temp	:= RIGHT( temp, LEN( temp ) - pos );
	pos		:= FIND( temp, rn ) - 1;
	sGeneral:= LEFT(temp, pos );
	pos		:= pos + LEN( rn );
	temp	:= RIGHT( temp, LEN( temp ) - pos );
	pos		:= FIND( temp, rn ) - 1;
	IF pos = -1 THEN
		pos := LEN( temp );
	END_IF
	sWork	:= LEFT(temp, pos );
	
	countStart.value	:= TO_REAL( sstart );
	countNO.value		:= TO_REAL( sNO );
	countAO.value		:= TO_REAL( sAO );
	
	generalOpTime.value	:= TO_REAL( sGeneral );
	workOpTime.value	:= TO_REAL( sWork );
	
	Read	:= TRUE;
END_IF

IF countFile.xError THEN
	err		:= countFile.eError;
	Read	:= TRUE;
END_IF
                        
END_METHOD

METHOD PRIVATE OpTime : BOOL
VAR
	cycle		: REAL;		// цикл вызова в часах
	currentTime	: UDINT;
END_VAR
VAR CONSTANT
	hour_ms	: REAL := 60_000.0 * 60.0;
END_VAR
                          currentTime	:= Util.SysTimeRtc.SysTimeGetMs();
cycle		:= TO_REAL( currentTime - oldTime ) / hour_ms;

generalOpTime.set_value	:= generalOpTime.value + cycle * TO_BYTE( isStarted );
workOpTime.set_value	:= workOpTime.value + cycle * TO_BYTE( work );

oldTime	:= Util.SysTimeRtc.SysTimeGetMs();
                        
END_METHOD
END_FUNCTION_BLOCK

// класс расчёта итоговой величина параметра по двум входным значениям
// Chekmarev 24.04.2025
//  0.0.01
// коэффициенты с 
FUNCTION_BLOCK TFreqRotorHandler
VAR_INPUT
	ch		: ARRAY[1..2] OF REAL; // измеряемые каналы
	minVal	: REAL	:= 100.0;
	maxVal	: REAL;
	flt_prm	: BOOL := TRUE;	// разрешение на расчёт неисправности
	disbal_Ch	: REAL := 100.0; // максимальный дисбаланс между каналами
	disbal_t: REAL	:= 0.16;// время расчёта дисбаланса, сек
	ucvV	: REAL	:= 500;	// максимальное изменение входной величины за цикл
	deblock	: BOOL;			// деблокировка
END_VAR
VAR_OUTPUT
	flt		: ARRAY[1..2] OF BOOL;	// отказ каналов по диапазону
	fltUcv	: ARRAY[1..2] OF BOOL;	// отказ каналов по скорости изменения
	disbal	: BOOL;
END_VAR
VAR_IN_OUT
	out		: Tacpar;
END_VAR
VAR
	oldVal	: ARRAY[1..2] OF REAL;
	disbalTmr	: TON;	// таймер дисбаланса
	ucvTmr		: ARRAY[1..2] OF TOF;	// таймеры удержки признака высокой скорости изменения
END_VAR
VAR CONSTANT
	ms_to_s	: UINT 	:= 1_000;
	PTucvTmr: TIME	:= T#30S;	// время удержания ПС по скорости изменения входного значения
END_VAR

                    flt_prm := flt_prm AND NOT deblock;

flt[1]	:= flt_prm AND ( ch[1] < minVal OR ch[1] > maxVal );
flt[2]	:= flt_prm AND ( ch[2] < minVal OR ch[2] > maxVal );

ucvTmr[1]( IN := flt_prm AND ABS( oldVal[1] - ch[1] ) > ucvV, PT := PTucvTmr );
ucvTmr[2]( IN := flt_prm AND ABS( oldVal[2] - ch[2] ) > ucvV, PT := PTucvTmr );

fltUcv[1] := ucvTmr[1].Q;
fltUcv[2] := ucvTmr[2].Q;

out.flt	:= ( flt[1] OR fltUcv[1] ) AND ( flt[2] OR fltUcv[2] );

IF ( ch[1] > ch[2] ) AND NOT ( flt[1] OR fltUcv[1] ) THEN
	out.in_value := ch[1];
	ELSIF NOT ( flt[2] OR fltUcv[2] ) THEN
	out.in_value := ch[2];
END_IF

disbalTmr (IN := flt_prm AND ( ABS( ch[1] - ch[2] ) > disbal_Ch ), PT := TO_TIME ( disbal_t * ms_to_s ));
disbal := disbalTmr.Q;

oldval[1] := ch[1];
oldVal[2] := ch[2];
                  
END_FUNCTION_BLOCK

// Контроль взвода защит на режимах
// Chekmarev
FUNCTION ShCntrl : BOOL
VAR
	shAlways	: BOOL;
	shInGas		: BOOL;
	shInWork	: BOOL;
	shOthers	: BOOL;
END_VAR

                    shAlways	:= 	crs.AO_BA.armed AND
				crs.AO_PRU.armed AND
				crs.AS_Av.armed AND
				crs.BEAO.armed AND
				crs.btn_AObs.armed AND
				crs.btn_AOss.armed AND
				crs.BZA_alr.armed AND
				crs.Chip_outD.armed AND
				crs.Fire_flt.armed AND
				crs.Fire_OD.armed AND
				crs.Nst_flt.armed AND
				crs.Nst_HH.armed AND
				crs.Ntk_Av_HH.armed AND
				crs.Ntk_flt.armed AND
				crs.Pa_out14_HH.armed  AND
				crs.SurgeD.armed AND
				crs.Tg_inST_HH.armed AND
				crs.Tg_inSTflt.armed AND
				crs.Tm_outD_HH.armed AND
				crs.Vs_D_Av.armed AND
				crs.Vsst_HH.armed AND
				crs.Vstk_HH.armed AND
				crs.Zs_Nl.armed ;
shInGas		:=	crs.dPmg_LL.armed AND tch.Gas_N.value OR NOT tch.Gas_N.value;
shInWork	:=( crs.Causeless_KR1_off.armed AND
				crs.Causeless_KR2_off.armed AND
				crs.Causeless_KR6_off.armed AND
				crs.KPV15_wOpen.armed AND 
				crs.Pm_ST_An.armed AND
				crs.Pm_TK_An.armed AND tch.GTDwork.value OR NOT tch.GTDwork.value ) AND
			  (	crs.Causeless_SK.armed AND
				crs.DGdistort.armed AND
				crs.KPV234_wOpen.armed AND
				crs.Pm_N_An.armed AND
				crs.Pm_SAR_An.armed AND
				crs.Ptg_inDG_An.armed AND
				crs.Ptg_inTRK_LL.armed AND
				crs.Tg1_inSTdistort_HH.armed AND
				crs.Tg2_inSTdistort_HH.armed AND
				crs.Tg3_inSTdistort_HH.armed AND
				crs.Tg4_inSTdistort_HH.armed AND
				crs.Tg5_inSTdistort_HH.armed AND
				crs.Tg6_inSTdistort_HH.armed AND ( tch.GTDHeat.value OR tch.GTDwork.value OR tch.GTDcool.value ) OR ( NOT tch.GTDHeat.value AND NOT tch.GTDwork.value AND NOT tch.GTDcool.value ));
shOthers	:=	crs.BZA_ready_2.armed AND
				crs.Causeless_KR10_11.armed AND
				crs.dP_F_Pv.armed AND
				crs.KPV15_nOpen.armed AND
				crs.Kr6_off_start.armed AND
				crs.nIgnition.armed AND	
				crs.Ntk_nBoost.armed AND
				crs.Pg_InKR13.armed AND
				crs.Pm_Starter_An.armed AND
				crs.Pm_Starter_Av.armed;

ShCntrl	:= shAlways AND shInGas AND shInWork;
                  
END_FUNCTION

PROGRAM PRG_IMIT
VAR
END_VAR

                    IF imitGPA.imit_on THEN
		GVL_IMIT.imitEngine(
		Tatm:= 15.0, 
		setDG1:= am.DG.set, 
		starter:= am.Kr11.isON AND am.Kr10.isOFF AND am.Kr13.on, 
		tuns:= ADR( GVL_IMIT.imitTuns ) 
		//posDG1=> , 
	);  
	
  	aipar.Ntk_1.sim_value := GVL_IMIT.imitEngine.Nvd;    
  	aipar.Ntk_2.sim_value := GVL_IMIT.imitEngine.Nvd;    
  	aipar.Nst_1.sim_value := GVL_IMIT.imitEngine.Nst;    
  	aipar.Nst_2.sim_value := GVL_IMIT.imitEngine.Nst;    
	aipar.Pa_out14.sim_value := GVL_IMIT.imitEngine.Pk;	
  	aipar.Tg_inST_1.sim_value := GVL_IMIT.imitEngine.Tst;  
  	aipar.Tg_inST_2.sim_value := GVL_IMIT.imitEngine.Tst;  
  	aipar.Tg_inST_3.sim_value := GVL_IMIT.imitEngine.Tst;  
  	aipar.Tg_inST_4.sim_value := GVL_IMIT.imitEngine.Tst;  
  	aipar.Tg_inST_5.sim_value := GVL_IMIT.imitEngine.Tst;  
  	aipar.Tg_inST_6.sim_value := GVL_IMIT.imitEngine.Tst;  
END_IF
                  
END_PROGRAM

PROGRAM HAND_DIAGN

                    UPD1_A1_1();
                  

ACTION UPD1_A1_1:
                        PsDiagn.PROXY_DI_16_012(MODULE := UPD1_A1_DI1, DATA := MODULE_UPD1_A1_DI1);
PsDiagn.PROXY_DI_16_012(MODULE := UPD1_A1_DI2, DATA := MODULE_UPD1_A1_DI2);
PsDiagn.PROXY_DI_16_012(MODULE := UPD1_A1_DI3, DATA := MODULE_UPD1_A1_DI3);
                      
END_ACTION
END_PROGRAM

{region INFO}
(*
 Назначение: Используется для сброса всех VAR_STAT сигнализаций
 Автор:  /Andrey/ 24.06.2025 16:50:31
 Версия: v00.00.22
 Проект: KA107__GPA2
*)
{endregion}
FUNCTION reset_alarm_var_stat : BOOL
VAR_INPUT
END_VAR

                    //Сбрасываем обобщенные сигнализации
//По типу и подсистемам в 0, потому что при сработке они выставляются в 1
crs.common.type_aggregated := crs.common.subsystem_aggregated := 0;
//По взводу защит все биты в 1, потому что при отсутствии взвода они сбрасываются в 0
crs.common.arm_aggregated := 16#FFFFFFFF;

//По типу биты 1-3 в 0 (для alr, lmt и trs, потому что при сработке они выставляются в 1), 4 и 5 в 1 (для ppu, потому что при сработке они сбрасываются в 0)
alr.common.type_aggregated := 2#110000;
//Для типов alr, lmt и trs по подсистемам все биты в 0, потому что при сработке они выставляются в 1
alr.common.subsystem_aggregated[1] := alr.common.subsystem_aggregated[2] := alr.common.subsystem_aggregated[3] := 0;
//Для ППУ по подсистемам все биты в 1, потому что при сработке они сбрасываются в 0
alr.common.subsystem_aggregated[4] := alr.common.subsystem_aggregated[5] := 16#FFFFFFFF;

                  
END_FUNCTION

{region INFO}
(*
 Назначение: Используется для сброса всех VAR_STAT входов/выходов
 Автор:  /Andrey/ 16.07.2025 17:15:05
 Версия: v00.00.01
 Проект: KA107
*)
{endregion}
FUNCTION reset_io_var_stat : BOOL
VAR_INPUT
END_VAR

                    //Сбрасываем для aipar
aipar.common.flt_aggregated := FALSE;
aipar.common.sim_aggregated := FALSE;
aipar.common.ucv_active := FALSE;

//Сбрасываем для aopar
aopar.common.flt_aggregated := FALSE;
aopar.common.sim_aggregated := FALSE;

//Сбрасываем для dipar
dipar.common.flt_aggregated := FALSE;
dipar.common.sim_aggregated := FALSE;

//Сбрасываем для dopar
dopar.common.flt_aggregated := FALSE;
dopar.common.sim_aggregated := FALSE;

                  
END_FUNCTION

{region INFO}
(*
 Назначение: Используется для сброса всех VAR_STAT ИМов
 Автор:  /Разработчик/ 08.08.2025 8:32:24
 Версия: v00.01.00
 Проект: KA107
*)
{endregion}
FUNCTION reset_am_var_stat : BOOL

                    am.common.flt_subsystem := 0;

                  
END_FUNCTION

// Используется для агрегации сигналов ИМов по подсистемам
FUNCTION aggregation_alarms : BOOL

                    
// crs
// Агрегация по типу
alg.AOss	:= crs.common.type_aggregated.1;
alg.AObs	:= crs.common.type_aggregated.2;


// ППУ
ppu.HR		:= ppu.common.type_aggregated.4;
ppu.GR		:= ppu.common.type_aggregated.5;

// Подсистемы
subsystem.EXT.aggregation_alarms( alr_common := alr.common, crs_common := crs.common );

subsystem.BD.aggregation_alarms( alr_common := alr.common, crs_common := crs.common );

subsystem.MSD.aggregation_alarms( alr_common := alr.common, crs_common := crs.common );

subsystem.VS.aggregation_alarms( alr_common := alr.common, crs_common := crs.common );

subsystem.AVOM.aggregation_alarms( alr_common := alr.common, crs_common := crs.common );

subsystem.BTG.aggregation_alarms( alr_common := alr.common, crs_common := crs.common );

subsystem.BPG.aggregation_alarms( alr_common := alr.common, crs_common := crs.common );

subsystem.POS.aggregation_alarms( alr_common := alr.common, crs_common := crs.common );

subsystem.BN.aggregation_alarms( alr_common := alr.common, crs_common := crs.common );

subsystem.BU.aggregation_alarms( alr_common := alr.common, crs_common := crs.common );

subsystem.GO.aggregation_alarms( alr_common := alr.common, crs_common := crs.common );
                  
END_FUNCTION

FUNCTION aggregation_am : BOOL

                    subsystem.EXT.AM_flt	:= am.common.flt_subsystem.1;

subsystem.BD.AM_flt		:= am.common.flt_subsystem.2;

subsystem.MSD.AM_flt	:= am.common.flt_subsystem.3;

subsystem.VS.AM_flt		:= am.common.flt_subsystem.4;

subsystem.AVOM.AM_flt	:= am.common.flt_subsystem.5;

subsystem.BTG.AM_flt	:= am.common.flt_subsystem.6;

subsystem.BPG.AM_flt	:= am.common.flt_subsystem.7;

subsystem.POS.AM_flt	:= am.common.flt_subsystem.8;

subsystem.BN.AM_flt		:= am.common.flt_subsystem.9;

subsystem.BU.AM_flt		:= am.common.flt_subsystem.10;

subsystem.GO.AM_flt		:= am.common.flt_subsystem.11;
                  
END_FUNCTION

FUNCTION ALG_BU_Link : BOOL

                    subsystem.BU();
                  
END_FUNCTION

FUNCTION ALG_VOU_Link : BOOL

                    subsystem.POS();
                  
END_FUNCTION

CONFIGURATION GPA2_SAU
  RESOURCE Application ON PLC
(* global variable list GVL_DIAGN *)
{attribute 'symbol' := 'readwrite'}
VAR_GLOBAL
	//Флаг активности ПЛК
	IS_ACTIVE: BOOL;
	//Активность ПЛК А
	IS_CPU_A: BOOL;
	//Активность ПЛК Б
	IS_CPU_B: BOOL;

	MODULE_UCP1_A1_ST1: PsDiagn.MODULE_ST_XX_X1X;
	MODULE_UCP1_A1_PP1: PsDiagn.MODULE_PP_00_XXX;
	MODULE_UCP1_A1_CU1: PsDiagn.MODULE_CU_XX_XXX;
	MODULE_UCP1_A1_FI1: PsDiagn.MODULE_DA_03_021_L_FRQ;
	MODULE_UCP1_A1_FI2: PsDiagn.MODULE_DA_03_021_L_FRQ;
	MODULE_UCP1_A1_AI1: PsDiagn.MODULE_AI_08_052;
	MODULE_UCP1_A1_AI2: PsDiagn.MODULE_AI_08_052;
	MODULE_UCP1_A1_AI3: PsDiagn.MODULE_AI_08_052;
	MODULE_UCP1_A1_AI4: PsDiagn.MODULE_AI_08_031;
	MODULE_UCP1_A1_AI5: PsDiagn.MODULE_AI_08_031;
	MODULE_UCP1_A1_AI6: PsDiagn.MODULE_AI_08_031;
	MODULE_UCP1_A1_AI7: PsDiagn.MODULE_AI_08_031;
	MODULE_UCP1_A1_ST2: PsDiagn.MODULE_ST_XX_X2X;
	MODULE_UCP1_A2_ST1: PsDiagn.MODULE_ST_XX_X1X;
	MODULE_UCP1_A2_PP1: PsDiagn.MODULE_PP_00_XXX;
	MODULE_UCP1_A2_AO1: PsDiagn.MODULE_AO_08_031;
	MODULE_UCP1_A2_DI1: PsDiagn.MODULE_AI_16_011;
	MODULE_UCP1_A2_DI2: PsDiagn.MODULE_AI_16_011;
	MODULE_UCP1_A2_DI3: PsDiagn.MODULE_DI_32_011;
	MODULE_UCP1_A2_DO1: PsDiagn.MODULE_DO_32_012;
	MODULE_UCP1_A2_DI4: PsDiagn.MODULE_DI_32_011;
	MODULE_UCP1_A2_ST2: PsDiagn.MODULE_ST_XX_X2X;
	MODULE_UE1_A1_ST1: PsDiagn.MODULE_ST_XX_X1X;
	MODULE_UE1_A1_PP1: PsDiagn.MODULE_PP_00_XXX;
	MODULE_UE1_A1_DI1: PsDiagn.MODULE_AI_16_011;
	MODULE_UE1_A1_DI2: PsDiagn.MODULE_AI_16_011;
	MODULE_UE1_A1_DI3: PsDiagn.MODULE_AI_16_011;
	MODULE_UE1_A1_DI4: PsDiagn.MODULE_DI_32_011;
	MODULE_UE1_A1_DI5: PsDiagn.MODULE_DI_32_011;
	MODULE_UE1_A1_DO1: PsDiagn.MODULE_DO_32_012;
	MODULE_UE1_A1_DI6: PsDiagn.MODULE_DI_32_011;
	MODULE_UE1_A1_DO2: PsDiagn.MODULE_DO_32_012;
	MODULE_UE1_A1_DI7: PsDiagn.MODULE_DI_32_011;
	MODULE_UE1_A1_ST2: PsDiagn.MODULE_ST_XX_X2X;
END_VAR
(* global variable list SETPOINTS_PERSISTENT_b9f40513_edea_4730_822c_5ab1a3caf7be *)
VAR_GLOBAL RETAIN PERSISTENT
	PERSISTENT_EXIST: BOOL;
END_VAR
(* global variable list alr *)
{region INFO}
(*
 Назначение: Признаки срабатывания предупредительных сигнализаций
 Автор:  /Andrey/ 24.06.2025 16:50:31
 Версия: v00.00.22
 Проект: KA107__GPA2
*)
{endregion}
{attribute 'qualified_only'}
{attribute 'symbol' := 'read'}
VAR_GLOBAL
	{attribute 'symbol' := 'none'}
	common : Talarm; //Общий сигнал для VAR_STAT

	{attribute 'export' := '("archive":"True","name":"Кнопка ЭАО на ПРУ нажата сигнал 1 (НР)","alarm":("type":"alr","action":"нет"),"condition":("set":"TRUE","reset":"FALSE","active":"dipar.EAO_PRU_1.value"))'}
	EAO_PRU_1 : Talarm:= (subsystem_num := 1, type_num := 1); //Кнопка ЭАО на ПРУ нажата сигнал 1 (НР)//DI/Внешние источники
	{attribute 'export' := '("archive":"True","name":"Кнопка ЭАО на ПРУ нажата сигнал 2 (НЗ)","alarm":("type":"alr","action":"нет"),"condition":("set":"TRUE","reset":"FALSE","active":"dipar.EAO_PRU_2.value"))'}
	EAO_PRU_2 : Talarm:= (subsystem_num := 1, type_num := 1); //Кнопка ЭАО на ПРУ нажата сигнал 2 (НЗ)//DI/Внешние источники
	{attribute 'export' := '("archive":"True","name":"Кнопка ЭАО на ПРУ нажата сигнал 3 (НЗ)","alarm":("type":"alr","action":"нет"),"condition":("set":"TRUE","reset":"FALSE","active":"dipar.EAO_PRU_3.value"))'}
	EAO_PRU_3 : Talarm:= (subsystem_num := 1, type_num := 1); //Кнопка ЭАО на ПРУ нажата сигнал 3 (НЗ)//DI/Внешние источники
	{attribute 'export' := '("archive":"True","name":"Нет связи с ПРУ","alarm":("type":"alr","action":"нет"),"condition":("set":"TRUE","reset":"FALSE","active":"NOT PRU.Link"))'}
	PRU_noLink : Talarm:= (subsystem_num := 1, type_num := 1, pt := t#1s0ms); //Нет связи с ПРУ//ALG/Внешние источники
	{attribute 'export' := '("archive":"True","name":"Загазованность контейнеров выше нормы","alarm":("type":"alr","action":"ХР"),"condition":("set":"TRUE","reset":"FALSE","active":"dipar.Zagaz_OD_Pv.value"))'}
	Zagaz_OD_Pv : Talarm:= (subsystem_num := 2, type_num := 1, pt := t#1s0ms); //Загазованность контейнеров выше нормы//DI/Блок двигателя
	{attribute 'export' := '("archive":"True","name":"Повышенная вибрация двигателя","alarm":("type":"alr","action":"нет"),"condition":("set":"TRUE","reset":"FALSE","active":"dipar.Vs_D_Pv.value"))'}
	Vs_D_Pv : Talarm:= (subsystem_num := 2, type_num := 1, pt := t#1s0ms); //Повышенная вибрация двигателя//DI/Блок двигателя
	{attribute 'export' := '("archive":"True","name":"Повыш. Вибрация ТК","alarm":("type":"alr","action":"нет"),"condition":("set":"TRUE","reset":"FALSE","active":"aipar.Vstk.setpoint.H"))'}
	Vstk_H : Talarm:= (subsystem_num := 2, type_num := 1, pt := t#1s0ms); //Повыш. Вибрация ТК//> 50/Блок двигателя
	{attribute 'export' := '("archive":"True","name":"Повыш. Вибрация СТ","alarm":("type":"alr","action":"нет"),"condition":("set":"TRUE","reset":"FALSE","active":"aipar.Vsst.setpoint.H"))'}
	Vsst_H : Talarm:= (subsystem_num := 2, type_num := 1, pt := t#1s0ms); //Повыш. Вибрация СТ//> 50/Блок двигателя
	{attribute 'export' := '("archive":"True","name":"Сигнализатор обледенения","alarm":("type":"alr","action":"ГР"),"condition":("set":"TRUE","reset":"FALSE","active":"dipar.Ace_alr.value"))'}
	Ace_alr : Talarm:= (subsystem_num := 2, type_num := 1, pt := t#1s0ms); //Сигнализатор обледенения//DI/Блок двигателя
	{attribute 'export' := '("archive":"True","name":"КПВ не открыты на пуске","alarm":("type":"alr","action":"нет"),"condition":("set":"acpar.Ntk.value > 2000 AND acpar.Ntk.value < 4500 AND alg.start","reset":"acpar.Ntk.value > 4500 OR alg.AO","active":"NOT ( dipar.KPV2_ON.value AND dipar.KPV3_ON.value AND dipar.KPV4_ON.value AND dipar.KPV1_ON.value AND dipar.KPV5_ON.value )"))'}
	KPV_nOpen : Talarm:= (subsystem_num := 2, type_num := 1, pt := t#1s0ms); //КПВ не открыты на пуске//DI/Блок двигателя
	{attribute 'export' := '("archive":"True","name":"КПВ234 не открыты","alarm":("type":"alr","action":"нет"),"condition":("set":"NOss.cmd_KPV234_On OR NObs.cmd_KPV234_On OR AOss.cmd_KPV234_On OR AObs.cmd_KPV234_On","reset":"acpar.Ntk.value < 2000","active":"NOT ( dipar.KPV2_ON.value AND dipar.KPV3_ON.value AND dipar.KPV4_ON.value )"))'}
	KPV234_nOpen : Talarm:= (subsystem_num := 2, type_num := 1, pt := t#1s0ms); //КПВ234 не открыты//ALG/Блок двигателя
	{attribute 'export' := '("archive":"True","name":"Повыш. Обороты СТ > 8500 об/мин","alarm":("type":"alr","action":"нет"),"condition":("set":"TRUE","reset":"FALSE","active":"acpar.Nst.setpoint.H"))'}
	Nst_H : Talarm:= (subsystem_num := 2, type_num := 1, pt := t#1s0ms); //Повыш. Обороты СТ > 8500 об/мин//> 8500 об/мин/Блок двигателя
	{attribute 'export' := '("archive":"True","name":"Высокая скорость изменения оборотов 1-ого канала ТК","alarm":("type":"alr","action":"нет"),"condition":("set":"TRUE","reset":"FALSE","active":"acpar_handler.handler.nTKcalc.fltUcv[1]"))'}
	Ntk_1_OV : Talarm:= (subsystem_num := 2, type_num := 1); //Высокая скорость изменения оборотов 1-ого канала ТК//ALG/Блок двигателя
	{attribute 'export' := '("archive":"True","name":"Высокая скорость изменения оборотов 2-ого канала ТК","alarm":("type":"alr","action":"нет"),"condition":("set":"TRUE","reset":"FALSE","active":"acpar_handler.handler.nTKcalc.fltUcv[2]"))'}
	Ntk_2_OV : Talarm:= (subsystem_num := 2, type_num := 1); //Высокая скорость изменения оборотов 2-ого канала ТК//ALG/Блок двигателя
	{attribute 'export' := '("archive":"True","name":"Значения оборотов 1-ого канала ТК не в диапазоне","alarm":("type":"alr","action":"нет"),"condition":("set":"TRUE","reset":"FALSE","active":"acpar_handler.handler.nTKcalc.flt[1]"))'}
	Ntk_1_UV : Talarm:= (subsystem_num := 2, type_num := 1); //Значения оборотов 1-ого канала ТК не в диапазоне//ALG/Блок двигателя
	{attribute 'export' := '("archive":"True","name":"Значения оборотов 2-ого канала ТК не в диапазоне","alarm":("type":"alr","action":"нет"),"condition":("set":"TRUE","reset":"FALSE","active":"acpar_handler.handler.nTKcalc.flt[2]"))'}
	Ntk_2_UV : Talarm:= (subsystem_num := 2, type_num := 1); //Значения оборотов 2-ого канала ТК не в диапазоне//ALG/Блок двигателя
	{attribute 'export' := '("archive":"True","name":"Значения оборотов 1-ого канала СТ не в диапазоне","alarm":("type":"alr","action":"нет"),"condition":("set":"TRUE","reset":"FALSE","active":"acpar_handler.handler.nSTcalc.flt[1]"))'}
	Nst_1_UV : Talarm:= (subsystem_num := 2, type_num := 1); //Значения оборотов 1-ого канала СТ не в диапазоне//ALG/Блок двигателя
	{attribute 'export' := '("archive":"True","name":"Значения оборотов 2-ого канала СТ не в диапазоне","alarm":("type":"alr","action":"нет"),"condition":("set":"TRUE","reset":"FALSE","active":"acpar_handler.handler.nSTcalc.flt[2]"))'}
	Nst_2_UV : Talarm:= (subsystem_num := 2, type_num := 1); //Значения оборотов 2-ого канала СТ не в диапазоне//ALG/Блок двигателя
	{attribute 'export' := '("archive":"True","name":"Высокая скорость изменения оборотов 1-ого канала СТ","alarm":("type":"alr","action":"нет"),"condition":("set":"TRUE","reset":"FALSE","active":"acpar_handler.handler.nSTcalc.fltUcv[1]"))'}
	Nst_1_OV : Talarm:= (subsystem_num := 2, type_num := 1); //Высокая скорость изменения оборотов 1-ого канала СТ//ALG/Блок двигателя
	{attribute 'export' := '("archive":"True","name":"Высокая скорость изменения оборотов 2-ого канала СТ","alarm":("type":"alr","action":"нет"),"condition":("set":"TRUE","reset":"FALSE","active":"acpar_handler.handler.nSTcalc.fltUcv[2]"))'}
	Nst_2_OV : Talarm:= (subsystem_num := 2, type_num := 1); //Высокая скорость изменения оборотов 2-ого канала СТ//ALG/Блок двигателя
	{attribute 'export' := '("archive":"True","name":"Повыш. Температура газа на входе СТ","alarm":("type":"alr","action":"нет"),"condition":("set":"TRUE","reset":"FALSE","active":"acpar.Tg_inST.setpoint.H"))'}
	Tg_inST_H : Talarm:= (subsystem_num := 2, type_num := 1); //Повыш. Температура газа на входе СТ//> 570 °С/Блок двигателя
	{attribute 'export' := '("archive":"True","name":"Нет сигнала: ТРК: готовность","alarm":("type":"alr","action":"ХР"),"condition":("set":"TRUE","reset":"FALSE","active":"NOT dipar.TRKready.value"))'}
	N_TRKready : Talarm:= (subsystem_num := 2, type_num := 1); //Нет сигнала: ТРК: готовность//Нет DI/Блок двигателя
	{attribute 'export' := '("archive":"True","name":"ТРК: авария","alarm":("type":"alr","action":"ХР"),"condition":("set":"TRUE","reset":"FALSE","active":"dipar.TRKalr.value"))'}
	TRKalr : Talarm:= (subsystem_num := 2, type_num := 1); //ТРК: авария//DI/Блок двигателя
	{attribute 'export' := '("archive":"True","name":"Контроль САУ не пройден","alarm":("type":"alr","action":"нет"),"condition":("set":"TRUE","reset":"FALSE","active":"check.tmrCancelPrm.Q"))'}
	nCheckSAU : Talarm:= (subsystem_num := 2, type_num := 1); //Контроль САУ не пройден//ALG/Блок двигателя
	{attribute 'export' := '("archive":"True","name":"Неисправность БЗА","alarm":("type":"alr","action":"нет"),"condition":("set":"tch.GTDWork.value","reset":"NOT tch.GTDWork.value","active":"NOT dipar.BZA_ready_1.value OR NOT dipar.BZA_ready_2.value"))'}
	BZA_flt : Talarm:= (subsystem_num := 2, type_num := 1); //Неисправность БЗА//ALG/Блок двигателя
	{attribute 'export' := '("archive":"True","name":"Пониж. Температура масла на входе двигателя","alarm":("type":"alr","action":"нет"),"condition":("set":"TRUE","reset":"FALSE","active":"aipar.Tm_inD.setpoint.L"))'}
	Tm_inD_L : Talarm:= (subsystem_num := 3, type_num := 1, pt := t#1s0ms); //Пониж. Температура масла на входе двигателя//< 40 °С/Маслосистема двигателя
	{attribute 'export' := '("archive":"True","name":"Уровень масла в МБД+Н минимальный","alarm":("type":"alr","action":"нет"),"condition":("set":"TRUE","reset":"FALSE","active":"dipar.Lm_MB_Pn.value"))'}
	Lm_MB_Pn : Talarm:= (subsystem_num := 3, type_num := 1, pt := t#1s0ms); //Уровень масла в МБД+Н минимальный//DI/Маслосистема двигателя
	{attribute 'export' := '("archive":"True","name":"Повыш. Температура масла на выходе АВОМД","alarm":("type":"alr","action":"нет"),"condition":("set":"TRUE","reset":"FALSE","active":"aipar.Tm_outAVOM.setpoint.H"))'}
	Tm_outAVOM_H : Talarm:= (subsystem_num := 5, type_num := 1, pt := t#1s0ms); //Повыш. Температура масла на выходе АВОМД//> 80 °С/Аппарат воздушного охлаждения масла двигателя
	{attribute 'export' := '("archive":"True","name":"Неисправность вентилятора 1 АВОМД","alarm":("type":"alr","action":"нет"),"condition":("set":"TRUE","reset":"FALSE","active":"am.Vn1_AVOM.flt"))'}
	Vn1_AVOM_flt : Talarm:= (subsystem_num := 5, type_num := 1, pt := t#1s0ms); //Неисправность вентилятора 1 АВОМД//DI/Аппарат воздушного охлаждения масла двигателя
	{attribute 'export' := '("archive":"True","name":"Неисправность вентилятора 2 АВОМД","alarm":("type":"alr","action":"нет"),"condition":("set":"TRUE","reset":"FALSE","active":"am.Vn2_AVOM.flt"))'}
	Vn2_AVOM_flt : Talarm:= (subsystem_num := 5, type_num := 1, pt := t#1s0ms); //Неисправность вентилятора 2 АВОМД//DI/Аппарат воздушного охлаждения масла двигателя
	{attribute 'export' := '("archive":"True","name":"Неисправность вентилятора 3 АВОМД","alarm":("type":"alr","action":"нет"),"condition":("set":"TRUE","reset":"FALSE","active":"am.Vn3_AVOM.flt"))'}
	Vn3_AVOM_flt : Talarm:= (subsystem_num := 5, type_num := 1, pt := t#1s0ms); //Неисправность вентилятора 3 АВОМД//DI/Аппарат воздушного охлаждения масла двигателя
	{attribute 'export' := '("archive":"True","name":"Неисправность вентилятора 4 АВОМД","alarm":("type":"alr","action":"нет"),"condition":("set":"TRUE","reset":"FALSE","active":"am.Vn4_AVOM.flt"))'}
	Vn4_AVOM_flt : Talarm:= (subsystem_num := 5, type_num := 1, pt := t#1s0ms); //Неисправность вентилятора 4 АВОМД//DI/Аппарат воздушного охлаждения масла двигателя
	{attribute 'export' := '("archive":"True","name":"Пониж. Давление топливного газа перед ТРК","alarm":("type":"alr","action":"нет"),"condition":("set":"alg.sh_TG","reset":"NOT alg.sh_TG","active":"aipar.Ptg_inTRK.setpoint.L"))'}
	Ptg_inTRK_L : Talarm:= (subsystem_num := 6, type_num := 1, pt := t#1s0ms); //Пониж. Давление топливного газа перед ТРК//< 20 кгс/см2/Блок топливного газа
	{attribute 'export' := '("archive":"True","name":"Повыш. Давление топливного газа перед ТРК","alarm":("type":"alr","action":"нет"),"condition":("set":"true","reset":"false","active":"aipar.Ptg_inTRK.setpoint.H"))'}
	Ptg_inTRK_H : Talarm:= (subsystem_num := 6, type_num := 1, pt := t#1s0ms); //Повыш. Давление топливного газа перед ТРК//> 27 кгс/см2/Блок топливного газа
	{attribute 'export' := '("archive":"True","name":"Давление газа перед дозатором газа Предупредительное","alarm":("type":"alr","action":"нет"),"condition":("set":"alg.sh_TG","reset":"NOT alg.sh_TG","active":"dipar.Ptg_inDG_Pn.value"))'}
	Ptg_inDG_Pn : Talarm:= (subsystem_num := 6, type_num := 1, pt := t#1s0ms); //Давление газа перед дозатором газа Предупредительное//DI/Блок топливного газа
	{attribute 'export' := '("archive":"True","name":"Перепад на сетке ВОУ","alarm":("type":"alr","action":"нет"),"condition":("set":"TRUE","reset":"FALSE","active":"dipar.Exh_VOU.value"))'}
	Exh_VOU : Talarm:= (subsystem_num := 8, type_num := 1, pt := t#1s0ms); //Перепад на сетке ВОУ//DI/Противообледенительная система и воздухоочистное устройство
	{attribute 'export' := '("archive":"True","name":"Опасность помпажа нагнетателя","alarm":("type":"alr","action":"нет"),"condition":("set":"TRUE","reset":"FALSE","active":"s_tunpar.ASprot.emergOpenBypass"))'}
	AS_Pv : Talarm:= (subsystem_num := 9, type_num := 1); //Опасность помпажа нагнетателя//ALG/Компрессорная установка/блок нагнетателя
	{attribute 'export' := '("archive":"True","name":"Пониж. Перепад давления “масло-газ”","alarm":("type":"alr","action":"нет"),"condition":("set":"alg.sh_dPmg","reset":"NOT alg.sh_dPmg","active":"aipar.dPmg.setpoint.L"))'}
	dPmg_L : Talarm:= (subsystem_num := 9, type_num := 1, pt := t#1s0ms); //Пониж. Перепад давления “масло-газ”//< 0.5 кгс/см2/Компрессорная установка/блок нагнетателя
	{attribute 'export' := '("archive":"True","name":"Уровень масла в МБУпл минимальный","alarm":("type":"alr","action":"нет"),"condition":("set":"TRUE","reset":"FALSE","active":"dipar.Lm_MBU_Pn.value"))'}
	Lm_MBU_Pn : Talarm:= (subsystem_num := 9, type_num := 1, pt := t#1s0ms); //Уровень масла в МБУпл минимальный//DI/Компрессорная установка/блок нагнетателя
	{attribute 'export' := '("archive":"True","name":"Повыш. Температура упорного подшипника Н","alarm":("type":"alr","action":"нет"),"condition":("set":"TRUE","reset":"FALSE","active":"aipar.Tup_N.setpoint.H"))'}
	Tup_N_H : Talarm:= (subsystem_num := 9, type_num := 1, pt := t#1s0ms); //Повыш. Температура упорного подшипника Н//> 80 °С/Компрессорная установка/блок нагнетателя
	{attribute 'export' := '("archive":"True","name":"Повыш. Температура опорного подшипника №1 Н","alarm":("type":"alr","action":"нет"),"condition":("set":"TRUE","reset":"FALSE","active":"aipar.Top_N_1.setpoint.H"))'}
	Top_N_1_H : Talarm:= (subsystem_num := 9, type_num := 1, pt := t#1s0ms); //Повыш. Температура опорного подшипника №1 Н//> 80 °С/Компрессорная установка/блок нагнетателя
	{attribute 'export' := '("archive":"True","name":"Повыш. Температура опорного подшипника №2 Н","alarm":("type":"alr","action":"нет"),"condition":("set":"TRUE","reset":"FALSE","active":"aipar.Top_N_2.setpoint.H"))'}
	Top_N_2_H : Talarm:= (subsystem_num := 9, type_num := 1, pt := t#1s0ms); //Повыш. Температура опорного подшипника №2 Н//> 80 °С/Компрессорная установка/блок нагнетателя
	{attribute 'export' := '("archive":"True","name":"Давление масла смазки Н предупредительная","alarm":("type":"alr","action":"нет"),"condition":("set":"NOT alg.V_000","reset":"alg.V_000","active":"dipar.Pm_N_Pn.value"))'}
	Pm_N_Pn : Talarm:= (subsystem_num := 9, type_num := 1, pt := t#1s0ms); //Давление масла смазки Н предупредительная//DI/Компрессорная установка/блок нагнетателя
	{attribute 'export' := '("archive":"True","name":"Нет сигнала: Предохранитель UCP1-XTFU1:1 питания модулей AO исправен","alarm":("type":"alr","action":"ХР"),"condition":("set":"TRUE","reset":"FALSE","active":"NOT dipar.Fuse_AO_UCP1.value"))'}
	N_Fuse_AO_UCP1 : Talarm:= (subsystem_num := 10, type_num := 1, pt := t#0s0ms); //Нет сигнала: Предохранитель UCP1-XTFU1:1 питания модулей AO исправен//Нет DI/Блок управления
	{attribute 'export' := '("archive":"True","name":"Нет сигнала: Предохранитель UCP1-XTFU1:2 питания модулей DO исправен","alarm":("type":"alr","action":"ХР"),"condition":("set":"TRUE","reset":"FALSE","active":"NOT dipar.Fuse_DO_UCP1.value"))'}
	N_Fuse_DO_UCP1 : Talarm:= (subsystem_num := 10, type_num := 1, pt := t#0s0ms); //Нет сигнала: Предохранитель UCP1-XTFU1:2 питания модулей DO исправен//Нет DI/Блок управления
	{attribute 'export' := '("archive":"True","name":"Нет сигнала: Предохранитель UCP1--XTFU6:1 питания датчиков температуры и влажности","alarm":("type":"alr","action":"ХР"),"condition":("set":"TRUE","reset":"FALSE","active":"NOT dipar.Fuse_Air_UCP1.value"))'}
	N_Fuse_Air_UCP1 : Talarm:= (subsystem_num := 10, type_num := 1, pt := t#0s0ms); //Нет сигнала: Предохранитель UCP1--XTFU6:1 питания датчиков температуры и влажности//Нет DI/Блок управления
	{attribute 'export' := '("archive":"True","name":"Нет сигнала: Предохранитель UE1-XTFU1:2 питания модулей DO исправен","alarm":("type":"alr","action":"ХР"),"condition":("set":"TRUE","reset":"FALSE","active":"NOT dipar.Fuse_DO_UE1.value"))'}
	N_Fuse_DO_UE1 : Talarm:= (subsystem_num := 10, type_num := 1, pt := t#0s0ms); //Нет сигнала: Предохранитель UE1-XTFU1:2 питания модулей DO исправен//Нет DI/Блок управления
	{attribute 'export' := '("archive":"True","name":"Перегрузка фильтра EV1 (Осн.)","alarm":("type":"alr","action":"ХР"),"condition":("set":"TRUE","reset":"FALSE","active":"dipar.EV1.value"))'}
	EV1 : Talarm:= (subsystem_num := 10, type_num := 1, pt := t#0s0ms); //Перегрузка фильтра EV1 (Осн.)//DI/Блок управления
	{attribute 'export' := '("archive":"True","name":"Перегрузка фильтра EV2 (Рез.)","alarm":("type":"alr","action":"ХР"),"condition":("set":"TRUE","reset":"FALSE","active":"dipar.EV2.value"))'}
	EV2 : Talarm:= (subsystem_num := 10, type_num := 1, pt := t#0s0ms); //Перегрузка фильтра EV2 (Рез.)//DI/Блок управления
	{attribute 'export' := '("archive":"True","name":"Нет сигнала: Контроль основного ввода питания (-KV1)","alarm":("type":"alr","action":"ХР"),"condition":("set":"TRUE","reset":"FALSE","active":"NOT dipar.U_main.value"))'}
	N_U_main : Talarm:= (subsystem_num := 10, type_num := 1, pt := t#0s0ms); //Нет сигнала: Контроль основного ввода питания (-KV1)//Нет DI/Блок управления
	{attribute 'export' := '("archive":"True","name":"Нет сигнала: Контроль резервного ввода питания (-KV2)","alarm":("type":"alr","action":"ХР"),"condition":("set":"TRUE","reset":"FALSE","active":"NOT dipar.U_res.value"))'}
	N_U_res : Talarm:= (subsystem_num := 10, type_num := 1, pt := t#0s0ms); //Нет сигнала: Контроль резервного ввода питания (-KV2)//Нет DI/Блок управления
	{attribute 'export' := '("archive":"True","name":"Контроль замыкания на землю питания PLC","alarm":("type":"alr","action":"нет"),"condition":("set":"TRUE","reset":"FALSE","active":"dipar.U_G_PLC.value"))'}
	U_G_PLC : Talarm:= (subsystem_num := 10, type_num := 1, pt := t#0s0ms); //Контроль замыкания на землю питания PLC//DI/Блок управления
	{attribute 'export' := '("archive":"True","name":"Контроль замыкания на землю питания AI","alarm":("type":"alr","action":"нет"),"condition":("set":"TRUE","reset":"FALSE","active":"dipar.U_G_AI.value"))'}
	U_G_AI : Talarm:= (subsystem_num := 10, type_num := 1, pt := t#0s0ms); //Контроль замыкания на землю питания AI//DI/Блок управления
	{attribute 'export' := '("archive":"True","name":"Контроль замыкания на землю питания DI","alarm":("type":"alr","action":"нет"),"condition":("set":"TRUE","reset":"FALSE","active":"dipar.U_G_DI.value"))'}
	U_G_DI : Talarm:= (subsystem_num := 10, type_num := 1, pt := t#0s0ms); //Контроль замыкания на землю питания DI//DI/Блок управления
	{attribute 'export' := '("archive":"True","name":"Контроль замыкания на землю питания БИЗ","alarm":("type":"alr","action":"нет"),"condition":("set":"TRUE","reset":"FALSE","active":"dipar.U_G_BIZ.value"))'}
	U_G_BIZ : Talarm:= (subsystem_num := 10, type_num := 1, pt := t#0s0ms); //Контроль замыкания на землю питания БИЗ//DI/Блок управления
	{attribute 'export' := '("archive":"True","name":"Нет сигнала: Контроль -AG1","alarm":("type":"alr","action":"ХР"),"condition":("set":"TRUE","reset":"FALSE","active":"NOT dipar.AG1.value"))'}
	N_AG1 : Talarm:= (subsystem_num := 10, type_num := 1, pt := t#0s0ms); //Нет сигнала: Контроль -AG1//Нет DI/Блок управления
	{attribute 'export' := '("archive":"True","name":"Нет сигнала: Контроль -AG2","alarm":("type":"alr","action":"ХР"),"condition":("set":"TRUE","reset":"FALSE","active":"NOT dipar.AG2.value"))'}
	N_AG2 : Talarm:= (subsystem_num := 10, type_num := 1, pt := t#0s0ms); //Нет сигнала: Контроль -AG2//Нет DI/Блок управления
	{attribute 'export' := '("archive":"True","name":"Нет сигнала: Контроль -AG3","alarm":("type":"alr","action":"ХР"),"condition":("set":"TRUE","reset":"FALSE","active":"NOT dipar.AG3.value"))'}
	N_AG3 : Talarm:= (subsystem_num := 10, type_num := 1, pt := t#0s0ms); //Нет сигнала: Контроль -AG3//Нет DI/Блок управления
	{attribute 'export' := '("archive":"True","name":"Нет сигнала: Контроль -AG4","alarm":("type":"alr","action":"ХР"),"condition":("set":"TRUE","reset":"FALSE","active":"NOT dipar.AG4.value"))'}
	N_AG4 : Talarm:= (subsystem_num := 10, type_num := 1, pt := t#0s0ms); //Нет сигнала: Контроль -AG4//Нет DI/Блок управления
	{attribute 'export' := '("archive":"True","name":"Нет сигнала: Контроль -AG9","alarm":("type":"alr","action":"ХР"),"condition":("set":"TRUE","reset":"FALSE","active":"NOT dipar.AG9.value"))'}
	N_AG9 : Talarm:= (subsystem_num := 10, type_num := 1, pt := t#0s0ms); //Нет сигнала: Контроль -AG9//Нет DI/Блок управления
	{attribute 'export' := '("archive":"True","name":"Нет сигнала: Контроль -AG10","alarm":("type":"alr","action":"ХР"),"condition":("set":"TRUE","reset":"FALSE","active":"NOT dipar.AG10.value"))'}
	N_AG10 : Talarm:= (subsystem_num := 10, type_num := 1, pt := t#0s0ms); //Нет сигнала: Контроль -AG10//Нет DI/Блок управления
	{attribute 'export' := '("archive":"True","name":"Нет сигнала: Контроль -AG15","alarm":("type":"alr","action":"ХР"),"condition":("set":"TRUE","reset":"FALSE","active":"NOT dipar.AG15.value"))'}
	N_AG15 : Talarm:= (subsystem_num := 10, type_num := 1, pt := t#0s0ms); //Нет сигнала: Контроль -AG15//Нет DI/Блок управления
	{attribute 'export' := '("archive":"True","name":"Нет сигнала: Контроль -AG16","alarm":("type":"alr","action":"ХР"),"condition":("set":"TRUE","reset":"FALSE","active":"NOT dipar.AG16.value"))'}
	N_AG16 : Talarm:= (subsystem_num := 10, type_num := 1, pt := t#0s0ms); //Нет сигнала: Контроль -AG16//Нет DI/Блок управления
	{attribute 'export' := '("archive":"True","name":"Нет сигнала: Контроль -AG5","alarm":("type":"alr","action":"ХР"),"condition":("set":"TRUE","reset":"FALSE","active":"NOT dipar.AG5.value"))'}
	N_AG5 : Talarm:= (subsystem_num := 10, type_num := 1, pt := t#0s0ms); //Нет сигнала: Контроль -AG5//Нет DI/Блок управления
	{attribute 'export' := '("archive":"True","name":"Нет сигнала: Контроль -AG6","alarm":("type":"alr","action":"ХР"),"condition":("set":"TRUE","reset":"FALSE","active":"NOT dipar.AG6.value"))'}
	N_AG6 : Talarm:= (subsystem_num := 10, type_num := 1, pt := t#0s0ms); //Нет сигнала: Контроль -AG6//Нет DI/Блок управления
	{attribute 'export' := '("archive":"True","name":"Нет сигнала: Контроль -AG8","alarm":("type":"alr","action":"ХР"),"condition":("set":"TRUE","reset":"FALSE","active":"NOT dipar.AG8.value"))'}
	N_AG8 : Talarm:= (subsystem_num := 10, type_num := 1, pt := t#0s0ms); //Нет сигнала: Контроль -AG8//Нет DI/Блок управления
	{attribute 'export' := '("archive":"True","name":"Нет сигнала: Контроль -AG17","alarm":("type":"alr","action":"ХР"),"condition":("set":"TRUE","reset":"FALSE","active":"NOT dipar.AG17.value"))'}
	N_AG17 : Talarm:= (subsystem_num := 10, type_num := 1, pt := t#0s0ms); //Нет сигнала: Контроль -AG17//Нет DI/Блок управления
	{attribute 'export' := '("archive":"True","name":"Нет сигнала: Контроль -AG18","alarm":("type":"alr","action":"ХР"),"condition":("set":"TRUE","reset":"FALSE","active":"NOT dipar.AG18.value"))'}
	N_AG18 : Talarm:= (subsystem_num := 10, type_num := 1, pt := t#0s0ms); //Нет сигнала: Контроль -AG18//Нет DI/Блок управления
	{attribute 'export' := '("archive":"True","name":"Нет сигнала: Контроль питания ПРУ","alarm":("type":"alr","action":"ХР"),"condition":("set":"TRUE","reset":"FALSE","active":"NOT dipar.U_PRU.value"))'}
	N_U_PRU : Talarm:= (subsystem_num := 10, type_num := 1, pt := t#0s0ms); //Нет сигнала: Контроль питания ПРУ//Нет DI/Блок управления
	{attribute 'export' := '("archive":"True","name":"Нет сигнала: Контроль питания ТРК осн.","alarm":("type":"alr","action":"ХР"),"condition":("set":"TRUE","reset":"FALSE","active":"NOT dipar.Utrk_main.value"))'}
	N_Utrk_main : Talarm:= (subsystem_num := 10, type_num := 1, pt := t#0s0ms); //Нет сигнала: Контроль питания ТРК осн.//Нет DI/Блок управления
	{attribute 'export' := '("archive":"True","name":"Контроль замыкания на землю питания ИМ","alarm":("type":"alr","action":"ХР"),"condition":("set":"TRUE","reset":"FALSE","active":"dipar.U_G_AM.value"))'}
	U_G_AM : Talarm:= (subsystem_num := 10, type_num := 1, pt := t#0s0ms); //Контроль замыкания на землю питания ИМ//DI/Блок управления
	{attribute 'export' := '("archive":"True","name":"Нет сигнала: Контроль питания AI","alarm":("type":"alr","action":"ХР"),"condition":("set":"TRUE","reset":"FALSE","active":"NOT dipar.U_AI.value"))'}
	N_U_AI : Talarm:= (subsystem_num := 10, type_num := 1, pt := t#0s0ms); //Нет сигнала: Контроль питания AI//Нет DI/Блок управления
	{attribute 'export' := '("archive":"True","name":"Нет сигнала: Контроль питания DI","alarm":("type":"alr","action":"ХР"),"condition":("set":"TRUE","reset":"FALSE","active":"NOT dipar.U_DI.value"))'}
	N_U_DI : Talarm:= (subsystem_num := 10, type_num := 1, pt := t#0s0ms); //Нет сигнала: Контроль питания DI//Нет DI/Блок управления
	{attribute 'export' := '("archive":"True","name":"Нет сигнала: Контроль питания БИЗ","alarm":("type":"alr","action":"ХР"),"condition":("set":"TRUE","reset":"FALSE","active":"NOT dipar.U_BIZ.value"))'}
	N_U_BIZ : Talarm:= (subsystem_num := 10, type_num := 1, pt := t#0s0ms); //Нет сигнала: Контроль питания БИЗ//Нет DI/Блок управления
	{attribute 'export' := '("archive":"True","name":"Нет сигнала: Контроль питания ИМ","alarm":("type":"alr","action":"ХР"),"condition":("set":"TRUE","reset":"FALSE","active":"NOT dipar.U_AM.value"))'}
	N_U_AM : Talarm:= (subsystem_num := 10, type_num := 1, pt := t#0s0ms); //Нет сигнала: Контроль питания ИМ//Нет DI/Блок управления
	{attribute 'export' := '("archive":"True","name":"Нет сигнала: Контроль питания аппаратуры вибрации, =24 В","alarm":("type":"alr","action":"ХР"),"condition":("set":"TRUE","reset":"FALSE","active":"NOT dipar.Uvs_24.value"))'}
	N_Uvs_24 : Talarm:= (subsystem_num := 10, type_num := 1, pt := t#0s0ms); //Нет сигнала: Контроль питания аппаратуры вибрации, =24 В//Нет DI/Блок управления
	{attribute 'export' := '("archive":"True","name":"Нет сигнала: Контроль питания дополнительного оборудования, =24В","alarm":("type":"alr","action":"ХР"),"condition":("set":"TRUE","reset":"FALSE","active":"NOT dipar.Uother_24.value"))'}
	N_Uother_24 : Talarm:= (subsystem_num := 10, type_num := 1, pt := t#0s0ms); //Нет сигнала: Контроль питания дополнительного оборудования, =24В//Нет DI/Блок управления
	{attribute 'export' := '("archive":"True","name":"Нет сигнала: Контроль питания ИМ2","alarm":("type":"alr","action":"ХР"),"condition":("set":"TRUE","reset":"FALSE","active":"NOT dipar.U_AM2.value"))'}
	N_U_AM2 : Talarm:= (subsystem_num := 10, type_num := 1, pt := t#0s0ms); //Нет сигнала: Контроль питания ИМ2//Нет DI/Блок управления
	{attribute 'export' := '("archive":"True","name":"Нет сигнала: Контроль питания ТРК рез.","alarm":("type":"alr","action":"ХР"),"condition":("set":"TRUE","reset":"FALSE","active":"NOT dipar.Utrk_res.value"))'}
	N_Utrk_res : Talarm:= (subsystem_num := 10, type_num := 1, pt := t#0s0ms); //Нет сигнала: Контроль питания ТРК рез.//Нет DI/Блок управления
	{attribute 'export' := '("archive":"True","name":"БЭО. Перегрузка фильтра EV3 (Осн. БЭО)","alarm":("type":"alr","action":"ХР"),"condition":("set":"TRUE","reset":"FALSE","active":"dipar.EV3.value"))'}
	EV3 : Talarm:= (subsystem_num := 10, type_num := 1, pt := t#0s0ms); //БЭО. Перегрузка фильтра EV3 (Осн. БЭО)//DI/Блок управления
	{attribute 'export' := '("archive":"True","name":"БЭО. Перегрузка фильтра EV4 (Рез. БЭО)","alarm":("type":"alr","action":"ХР"),"condition":("set":"TRUE","reset":"FALSE","active":"dipar.EV4.value"))'}
	EV4 : Talarm:= (subsystem_num := 10, type_num := 1, pt := t#0s0ms); //БЭО. Перегрузка фильтра EV4 (Рез. БЭО)//DI/Блок управления
	{attribute 'export' := '("archive":"True","name":"Нет сигнала: БЭО. Контроль основного ввода питания БЭО (-KV3)","alarm":("type":"alr","action":"ХР"),"condition":("set":"TRUE","reset":"FALSE","active":"NOT dipar.Ubeo_main.value"))'}
	N_Ubeo_main : Talarm:= (subsystem_num := 10, type_num := 1, pt := t#0s0ms); //Нет сигнала: БЭО. Контроль основного ввода питания БЭО (-KV3)//Нет DI/Блок управления
	{attribute 'export' := '("archive":"True","name":"Нет сигнала: БЭО. Контроль резервного ввода питания БЭО (-KV4)","alarm":("type":"alr","action":"ХР"),"condition":("set":"TRUE","reset":"FALSE","active":"NOT dipar.Ubeo_res.value"))'}
	N_Ubeo_res : Talarm:= (subsystem_num := 10, type_num := 1, pt := t#0s0ms); //Нет сигнала: БЭО. Контроль резервного ввода питания БЭО (-KV4)//Нет DI/Блок управления
	{attribute 'export' := '("archive":"True","name":"Нет сигнала: БЭО. Контроль -AG11","alarm":("type":"alr","action":"ХР"),"condition":("set":"TRUE","reset":"FALSE","active":"NOT dipar.AG11.value"))'}
	N_AG11 : Talarm:= (subsystem_num := 10, type_num := 1, pt := t#0s0ms); //Нет сигнала: БЭО. Контроль -AG11//Нет DI/Блок управления
	{attribute 'export' := '("archive":"True","name":"Нет сигнала: БЭО. Контроль -AG12","alarm":("type":"alr","action":"ХР"),"condition":("set":"TRUE","reset":"FALSE","active":"NOT dipar.AG12.value"))'}
	N_AG12 : Talarm:= (subsystem_num := 10, type_num := 1, pt := t#0s0ms); //Нет сигнала: БЭО. Контроль -AG12//Нет DI/Блок управления
	{attribute 'export' := '("archive":"True","name":"БЭО. Контроль замыкания на землю питания БЭО (-KR5)","alarm":("type":"alr","action":"ХР"),"condition":("set":"TRUE","reset":"FALSE","active":"dipar.U_G_KR5.value"))'}
	U_G_KR5 : Talarm:= (subsystem_num := 10, type_num := 1, pt := t#0s0ms); //БЭО. Контроль замыкания на землю питания БЭО (-KR5)//DI/Блок управления
	{attribute 'export' := '("archive":"True","name":"Нет сигнала: БЭО. Контроль питания кн. ЭАО","alarm":("type":"alr","action":"ХР"),"condition":("set":"TRUE","reset":"FALSE","active":"NOT dipar.U_KEAO.value"))'}
	N_U_KEAO : Talarm:= (subsystem_num := 10, type_num := 1, pt := t#0s0ms); //Нет сигнала: БЭО. Контроль питания кн. ЭАО//Нет DI/Блок управления
	{attribute 'export' := '("archive":"True","name":"Нет сигнала: БЭО. Контроль питания БЭО","alarm":("type":"alr","action":"ХР"),"condition":("set":"TRUE","reset":"FALSE","active":"NOT dipar.U_BEO.value"))'}
	N_U_BEO : Talarm:= (subsystem_num := 10, type_num := 1, pt := t#0s0ms); //Нет сигнала: БЭО. Контроль питания БЭО//Нет DI/Блок управления
	{attribute 'export' := '("archive":"True","name":"Нет сигнала: БЭО. Контроль питания БЗА","alarm":("type":"alr","action":"ХР"),"condition":("set":"TRUE","reset":"FALSE","active":"NOT dipar.U_BZA.value"))'}
	N_U_BZA : Talarm:= (subsystem_num := 10, type_num := 1, pt := t#0s0ms); //Нет сигнала: БЭО. Контроль питания БЗА//Нет DI/Блок управления
	{attribute 'export' := '("archive":"True","name":"Ошибка -AUO1","alarm":("type":"alr","action":"ХР"),"condition":("set":"TRUE","reset":"FALSE","active":"dipar.Err_AUO1.value"))'}
	Err_AUO1 : Talarm:= (subsystem_num := 10, type_num := 1, pt := t#0s0ms); //Ошибка -AUO1//DI/Блок управления
	{attribute 'export' := '("archive":"True","name":"Одна или более защит не взведены","alarm":("type":"alr","action":"нет"),"condition":("set":"TRUE","reset":"FALSE","active":"NOT alg.sh_cntrl"))'}
	shCntrl : Talarm:= (subsystem_num := 12, type_num := 1, pt := t#5s0ms); //Одна или более защит не взведены//ALG/Контроль защит
END_VAR
(* global variable list crs *)
{region INFO}
(*
 Назначение: Признаки срабатывания аварийных сигнализаций, приводящих к останову
 Автор:  /Andrey/ 24.06.2025 16:50:31
 Версия: v00.00.22
 Проект: KA107__GPA2
*)
{endregion}
{attribute 'qualified_only'}
{attribute 'symbol' := 'readwrite'}
VAR_GLOBAL
	{attribute 'symbol' := 'none'}
	common: Tcrs; //Общий сигнал для VAR_STAT

